LIN {X 0,Y 236.009,Z 217.756,A -85,B 0,C 180,E1 -19840.931,E2 -19840.931} C_VEL
LIN {X 0,Y 236.536,Z 220.925,A -85,B 0,C 180,E1 -19845.488,E2 -19845.488} C_VEL
LIN {X 0,Y 237.16,Z 224.354,A -85,B 0,C 180,E1 -19849.755,E2 -19849.755} C_VEL
LIN {X 0,Y 237.857,Z 228.006,A -85,B 0,C 180,E1 -19853.776,E2 -19853.776} C_VEL
LIN {X 0,Y 238.192,Z 230.1,A -85,B 0,C 180,E1 -19855.902,E2 -19855.902} C_VEL
LIN {X 0,Y 238.171,Z 231.141,A -85,B 0,C 180,E1 -19856.891,E2 -19856.891} C_VEL
LIN {X 0,Y 237.53,Z 232.457,A -85,B 0,C 180,E1 -19857.82,E2 -19857.82} C_VEL
LIN {X 0,Y 236.053,Z 234.265,A -85,B 0,C 180,E1 -19858.662,E2 -19858.662} C_VEL
LIN {X 0,Y 233.823,Z 237.363,A -85,B 0,C 180,E1 -19859.655,E2 -19859.655} C_VEL
LIN {X 0,Y 232.498,Z 240.8,A -85,B 0,C 180,E1 -19860.41,E2 -19860.41} C_VEL
LIN {X 0,Y 232.468,Z 243.65,A -85,B 0,C 180,E1 -19860.853,E2 -19860.853} C_VEL
LIN {X 0,Y 234.615,Z 253.264,A -85,B 0,C 180,E1 -19862.335,E2 -19862.335} C_VEL
LIN {X 0,Y 236.051,Z 263.876,A -85,B 0,C 180,E1 -19864.108,E2 -19864.108} C_VEL
LIN {X 0,Y 236.356,Z 273.236,A -85,B 0,C 180,E1 -19865.867,E2 -19865.867} C_VEL
LIN {X 0,Y 235.97,Z 280.551,A -85,B 0,C 180,E1 -19867.414,E2 -19867.414} C_VEL
LIN {X 0,Y 234.95,Z 287.098,A -85,B 0,C 180,E1 -19868.964,E2 -19868.964} C_VEL
LIN {X 0,Y 233.172,Z 293.307,A -85,B 0,C 180,E1 -19870.637,E2 -19870.637} C_VEL
LIN {X 0,Y 231.381,Z 298.539,A -85,B 0,C 180,E1 -19872.318,E2 -19872.318} C_VEL
LIN {X 0,Y 229.875,Z 302.919,A -85,B 0,C 180,E1 -19874.029,E2 -19874.029} C_VEL
LIN {X 0,Y 228.132,Z 308.12,A -85,B 0,C 180,E1 -19876.641,E2 -19876.641} C_VEL
LIN {X 0,Y 226.879,Z 311.977,A -85,B 0,C 180,E1 -19879.289,E2 -19879.289} C_VEL
LIN {X 0,Y 226.283,Z 313.766,A -85,B 0,C 180,E1 -19881.067,E2 -19881.067} C_VEL
LIN {X 0,Y 225.924,Z 315.065,A -85,B 0,C 180,E1 -19882.852,E2 -19882.852} C_VEL
LIN {X 0,Y 225.7,Z 316.017,A -85,B 0,C 180,E1 -19885.174,E2 -19885.174} C_VEL
LIN {X 0,Y 225.696,Z 316.253,A -85,B 0,C 180,E1 -19886.43,E2 -19886.43} C_VEL
LIN {X 0,Y 225.832,Z 316.034,A -85,B 0,C 180,E1 -19888.217,E2 -19888.217} C_VEL
LIN {X 0,Y 225.879,Z 315.278,A -85,B 0,C 180,E1 -19890,E2 -19890} C_VEL
LIN {X 0,Y 225.876,Z 314.017,A -85,B 0,C 180,E1 -19891.783,E2 -19891.783} C_VEL
LIN {X 0,Y 225.812,Z 311.128,A -85,B 0,C 180,E1 -19894.425,E2 -19894.425} C_VEL
LIN {X 0,Y 225.998,Z 306.803,A -85,B 0,C 180,E1 -19897.146,E2 -19897.146} C_VEL
LIN {X 0,Y 226.408,Z 301.952,A -85,B 0,C 180,E1 -19899.38,E2 -19899.38} C_VEL
LIN {X 0,Y 227.019,Z 295.755,A -85,B 0,C 180,E1 -19901.609,E2 -19901.609} C_VEL
LIN {X 0,Y 227.707,Z 289.678,A -85,B 0,C 180,E1 -19903.385,E2 -19903.385} C_VEL
LIN {X 0,Y 228.46,Z 283.285,A -85,B 0,C 180,E1 -19904.93,E2 -19904.93} C_VEL
LIN {X 0,Y 229.261,Z 278.016,A -85,B 0,C 180,E1 -19906.016,E2 -19906.016} C_VEL
LIN {X 0,Y 229.144,Z 270.13,A -85,B 0,C 180,E1 -19907.4,E2 -19907.4} C_VEL
LIN {X 0,Y 228.693,Z 261.091,A -85,B 0,C 180,E1 -19908.697,E2 -19908.697} C_VEL
LIN {X 0,Y 228.089,Z 252.419,A -85,B 0,C 180,E1 -19909.695,E2 -19909.695} C_VEL
LIN {X 0,Y 227.211,Z 241.832,A -85,B 0,C 180,E1 -19910.63,E2 -19910.63} C_VEL
LIN {X 0,Y 226.862,Z 237.785,A -85,B 0,C 180,E1 -19910.93,E2 -19910.93} C_VEL
LIN {X 0,Y 228.112,Z 230.392,A -85,B 0,C 180,E1 -19916.685,E2 -19916.685} C_VEL
LIN {X 0,Y 229.463,Z 224.432,A -85,B 0,C 180,E1 -19921.378,E2 -19921.378} C_VEL
LIN {X 0,Y 229.69,Z 223.191,A -85,B 0,C 180,E1 -19922.376,E2 -19922.376} C_VEL
LIN {X 0,Y 229.223,Z 219.34,A -85,B 0,C 180,E1 -19925.63,E2 -19925.63} C_VEL
LIN {X 0,Y 228.198,Z 214.067,A -85,B 0,C 180,E1 -19930.298,E2 -19930.298} C_VEL
LIN {X 0,Y 227.968,Z 212.904,A -85,B 0,C 180,E1 -19931.516,E2 -19931.516} C_VEL
LIN {X 0,Y 227.833,Z 212.914,A -85,B 0,C 180,E1 -19935.194,E2 -19935.194} C_VEL
LIN {X 0,Y 227.814,Z 212.918,A -85,B 0,C 180,E1 -19939.619,E2 -19939.619} C_VEL
LIN {X 0,Y 227.885,Z 212.91,A -85,B 0,C 180,E1 -19944.128,E2 -19944.128} C_VEL
LIN {X 0,Y 227.871,Z 212.913,A -85,B 0,C 180,E1 -19948.377,E2 -19948.377} C_VEL
LIN {X 0,Y 227.884,Z 212.907,A -85,B 0,C 180,E1 -19952.443,E2 -19952.443} C_VEL
LIN {X 0,Y 227.911,Z 212.907,A -85,B 0,C 180,E1 -19956.366,E2 -19956.366} C_VEL
LIN {X 0,Y 227.942,Z 212.901,A -85,B 0,C 180,E1 -19960.173,E2 -19960.173} C_VEL
LIN {X 0,Y 228.062,Z 212.889,A -85,B 0,C 180,E1 -19963.897,E2 -19963.897} C_VEL
LIN {X 0,Y 228.076,Z 212.888,A -85,B 0,C 180,E1 -19967.542,E2 -19967.542} C_VEL
LIN {X 0,Y 228.267,Z 212.861,A -85,B 0,C 180,E1 -19971.143,E2 -19971.143} C_VEL
LIN {X 0,Y 228.322,Z 212.855,A -85,B 0,C 180,E1 -19972.926,E2 -19972.926} C_VEL
LIN {X 0,Y 228.557,Z 212.822,A -85,B 0,C 180,E1 -19978.236,E2 -19978.236} C_VEL
LIN {X 0,Y 228.557,Z 212.826,A -85,B 0,C 180,E1 -19981.761,E2 -19981.761} C_VEL
LIN {X 0,Y 228.321,Z 212.856,A -85,B 0,C 180,E1 -19987.071,E2 -19987.071} C_VEL
LIN {X 0,Y 228.144,Z 212.879,A -85,B 0,C 180,E1 -19990.65,E2 -19990.65} C_VEL
LIN {X 0,Y 228.036,Z 212.89,A -85,B 0,C 180,E1 -19994.272,E2 -19994.272} C_VEL
LIN {X 0,Y 227.952,Z 212.901,A -85,B 0,C 180,E1 -19997.956,E2 -19997.956} C_VEL
LIN {X 0,Y 227.915,Z 212.907,A -85,B 0,C 180,E1 -20002.318,E2 -20002.318} C_VEL
LIN {X 0,Y 227.942,Z 212.905,A -85,B 0,C 180,E1 -20006.601,E2 -20006.601} C_VEL
LIN {X 0,Y 227.908,Z 212.908,A -85,B 0,C 180,E1 -20010.294,E2 -20010.294} C_VEL
LIN {X 0,Y 227.888,Z 212.908,A -85,B 0,C 180,E1 -20013.716,E2 -20013.716} C_VEL
LIN {X 0,Y 227.867,Z 212.914,A -85,B 0,C 180,E1 -20018.084,E2 -20018.084} C_VEL
LIN {X 0,Y 227.81,Z 212.919,A -85,B 0,C 180,E1 -20022.74,E2 -20022.74} C_VEL
LIN {X 0,Y 227.807,Z 212.918,A -85,B 0,C 180,E1 -20027.256,E2 -20027.256} C_VEL
LIN {X 0,Y 227.84,Z 212.918,A -85,B 0,C 180,E1 -20031.907,E2 -20031.907} C_VEL
LIN {X 0,Y 227.877,Z 212.907,A -85,B 0,C 180,E1 -20036.375,E2 -20036.375} C_VEL
LIN {X 0,Y 227.915,Z 212.906,A -85,B 0,C 180,E1 -20040.437,E2 -20040.437} C_VEL
LIN {X 0,Y 227.923,Z 212.902,A -85,B 0,C 180,E1 -20044.425,E2 -20044.425} C_VEL
LIN {X 0,Y 227.956,Z 212.9,A -85,B 0,C 180,E1 -20048.286,E2 -20048.286} C_VEL
LIN {X 0,Y 228.028,Z 212.891,A -85,B 0,C 180,E1 -20052.825,E2 -20052.825} C_VEL
LIN {X 0,Y 228.088,Z 212.885,A -85,B 0,C 180,E1 -20057.544,E2 -20057.544} C_VEL
LIN {X 0,Y 228.299,Z 212.857,A -85,B 0,C 180,E1 -20061.145,E2 -20061.145} C_VEL
LIN {X 0,Y 228.348,Z 212.852,A -85,B 0,C 180,E1 -20062.928,E2 -20062.928} C_VEL
LIN {X 0,Y 228.547,Z 212.827,A -85,B 0,C 180,E1 -20068.237,E2 -20068.237} C_VEL
LIN {X 0,Y 228.547,Z 212.825,A -85,B 0,C 180,E1 -20071.762,E2 -20071.762} C_VEL
LIN {X 0,Y 228.342,Z 212.851,A -85,B 0,C 180,E1 -20077.072,E2 -20077.072} C_VEL
LIN {X 0,Y 228.069,Z 212.889,A -85,B 0,C 180,E1 -20080.654,E2 -20080.654} C_VEL
LIN {X 0,Y 227.568,Z 212.948,A -85,B 0,C 180,E1 -20085.219,E2 -20085.219} C_VEL
LIN {X 0,Y 227.387,Z 213.262,A -85,B 0,C 180,E1 -20086.151,E2 -20086.151} C_VEL
LIN {X 0,Y 226.732,Z 218.382,A -85,B 0,C 180,E1 -20091.836,E2 -20091.836} C_VEL
LIN {X 0,Y 226.515,Z 221.365,A -85,B 0,C 180,E1 -20095.069,E2 -20095.069} C_VEL
LIN {X 0,Y 228.367,Z 233.039,A -85,B 0,C 180,E1 -20096.142,E2 -20096.142} C_VEL
LIN {X 0,Y 229.539,Z 241.029,A -85,B 0,C 180,E1 -20097.094,E2 -20097.094} C_VEL
LIN {X 0,Y 230.39,Z 248.198,A -85,B 0,C 180,E1 -20098.118,E2 -20098.118} C_VEL
LIN {X 0,Y 230.632,Z 251.482,A -85,B 0,C 180,E1 -20098.632,E2 -20098.632} C_VEL
LIN {X 0,Y 229.569,Z 260.933,A -85,B 0,C 180,E1 -20100.34,E2 -20100.34} C_VEL
LIN {X 0,Y 228.561,Z 268.372,A -85,B 0,C 180,E1 -20102.033,E2 -20102.033} C_VEL
LIN {X 0,Y 227.799,Z 274.475,A -85,B 0,C 180,E1 -20103.733,E2 -20103.733} C_VEL
LIN {X 0,Y 226.95,Z 281.168,A -85,B 0,C 180,E1 -20106.042,E2 -20106.042} C_VEL
LIN {X 0,Y 226.266,Z 286.441,A -85,B 0,C 180,E1 -20108.405,E2 -20108.405} C_VEL
LIN {X 0,Y 225.798,Z 290.425,A -85,B 0,C 180,E1 -20110.815,E2 -20110.815} C_VEL
LIN {X 0,Y 225.52,Z 294.234,A -85,B 0,C 180,E1 -20114.215,E2 -20114.215} C_VEL
LIN {X 0,Y 225.654,Z 295.712,A -85,B 0,C 180,E1 -20116.752,E2 -20116.752} C_VEL
LIN {X 0,Y 226.034,Z 296.092,A -85,B 0,C 180,E1 -20119.238,E2 -20119.238} C_VEL
LIN {X 0,Y 226.727,Z 295.476,A -85,B 0,C 180,E1 -20121.69,E2 -20121.69} C_VEL
LIN {X 0,Y 227.729,Z 293.88,A -85,B 0,C 180,E1 -20124.103,E2 -20124.103} C_VEL
LIN {X 0,Y 228.965,Z 291.312,A -85,B 0,C 180,E1 -20126.463,E2 -20126.463} C_VEL
LIN {X 0,Y 230.971,Z 286.624,A -85,B 0,C 180,E1 -20129.36,E2 -20129.36} C_VEL
LIN {X 0,Y 233.004,Z 281.169,A -85,B 0,C 180,E1 -20131.726,E2 -20131.726} C_VEL
LIN {X 0,Y 234.562,Z 276.653,A -85,B 0,C 180,E1 -20133.295,E2 -20133.295} C_VEL
LIN {X 0,Y 236.617,Z 270.345,A -85,B 0,C 180,E1 -20135.063,E2 -20135.063} C_VEL
LIN {X 0,Y 238.257,Z 264.393,A -85,B 0,C 180,E1 -20136.444,E2 -20136.444} C_VEL
LIN {X 0,Y 237.992,Z 256.862,A -85,B 0,C 180,E1 -20138.222,E2 -20138.222} C_VEL
LIN {X 0,Y 236.795,Z 248.433,A -85,B 0,C 180,E1 -20140.045,E2 -20140.045} C_VEL
LIN {X 0,Y 234.593,Z 239.575,A -85,B 0,C 180,E1 -20141.832,E2 -20141.832} C_VEL
LIN {X 0,Y 230.936,Z 229.569,A -85,B 0,C 180,E1 -20143.742,E2 -20143.742} C_VEL
LIN {X 0,Y 229.933,Z 227.141,A -85,B 0,C 180,E1 -20144.205,E2 -20144.205} C_VEL
LIN {X 0,Y 228.809,Z 223.879,A -85,B 0,C 180,E1 -20144.81,E2 -20144.81} C_VEL
LIN {X 0,Y 229.302,Z 220.946,A -85,B 0,C 180,E1 -20149.405,E2 -20149.405} C_VEL
LIN {X 0,Y 229.234,Z 218.974,A -85,B 0,C 180,E1 -20152.957,E2 -20152.957} C_VEL
LIN {X 0,Y 229.128,Z 216.447,A -85,B 0,C 180,E1 -20158.244,E2 -20158.244} C_VEL
LIN {X 0,Y 229.155,Z 215.721,A -85,B 0,C 180,E1 -20160.002,E2 -20160.002} C_VEL
LIN {X 0,Y 228.593,Z 214.576,A -85,B 0,C 180,E1 -20163.527,E2 -20163.527} C_VEL
LIN {X 0,Y 228.444,Z 213.575,A -85,B 0,C 180,E1 -20167.07,E2 -20167.07} C_VEL
LIN {X 0,Y 228.147,Z 212.893,A -85,B 0,C 180,E1 -20170.653,E2 -20170.653} C_VEL
LIN {X 0,Y 228.066,Z 212.889,A -85,B 0,C 180,E1 -20174.273,E2 -20174.273} C_VEL
LIN {X 0,Y 228.006,Z 212.896,A -85,B 0,C 180,E1 -20177.954,E2 -20177.954} C_VEL
LIN {X 0,Y 227.933,Z 212.905,A -85,B 0,C 180,E1 -20182.331,E2 -20182.331} C_VEL
LIN {X 0,Y 228.046,Z 213.463,A -85,B 0,C 180,E1 -20186.655,E2 -20186.655} C_VEL
LIN {X 0,Y 228.219,Z 214.544,A -85,B 0,C 180,E1 -20190.429,E2 -20190.429} C_VEL
LIN {X 0,Y 228.472,Z 215.839,A -85,B 0,C 180,E1 -20193.846,E2 -20193.846} C_VEL
LIN {X 0,Y 228.798,Z 217.794,A -85,B 0,C 180,E1 -20197.905,E2 -20197.905} C_VEL
LIN {X 0,Y 229.049,Z 219.022,A -85,B 0,C 180,E1 -20200.119,E2 -20200.119} C_VEL
LIN {X 0,Y 229.547,Z 222.05,A -85,B 0,C 180,E1 -20204.765,E2 -20204.765} C_VEL
LIN {X 0,Y 229.969,Z 224.284,A -85,B 0,C 180,E1 -20207.753,E2 -20207.753} C_VEL
LIN {X 0,Y 230.669,Z 228.186,A -85,B 0,C 180,E1 -20212.39,E2 -20212.39} C_VEL
LIN {X 0,Y 231.105,Z 230.795,A -85,B 0,C 180,E1 -20215.195,E2 -20215.195} C_VEL
LIN {X 0,Y 231.186,Z 232.43,A -85,B 0,C 180,E1 -20216.826,E2 -20216.826} C_VEL
LIN {X 0,Y 230.299,Z 235.782,A -85,B 0,C 180,E1 -20219.736,E2 -20219.736} C_VEL
LIN {X 0,Y 231.26,Z 239.321,A -85,B 0,C 180,E1 -20220.208,E2 -20220.208} C_VEL
LIN {X 0,Y 232.468,Z 243.65,A -85,B 0,C 180,E1 -20220.853,E2 -20220.853} C_VEL
LIN {X 0,Y 232.865,Z 248.996,A -85,B 0,C 180,E1 -20221.485,E2 -20221.485} C_VEL
LIN {X 0,Y 231.841,Z 258.038,A -85,B 0,C 180,E1 -20222.481,E2 -20222.481} C_VEL
LIN {X 0,Y 230.335,Z 266.707,A -85,B 0,C 180,E1 -20223.644,E2 -20223.644} C_VEL
LIN {X 0,Y 229.968,Z 271.47,A -85,B 0,C 180,E1 -20224.529,E2 -20224.529} C_VEL
LIN {X 0,Y 229.709,Z 278.727,A -85,B 0,C 180,E1 -20226.085,E2 -20226.085} C_VEL
LIN {X 0,Y 228.639,Z 286.775,A -85,B 0,C 180,E1 -20228.06,E2 -20228.06} C_VEL
LIN {X 0,Y 227.007,Z 292.445,A -85,B 0,C 180,E1 -20229.617,E2 -20229.617} C_VEL
LIN {X 0,Y 225.068,Z 297.746,A -85,B 0,C 180,E1 -20231.333,E2 -20231.333} C_VEL
LIN {X 0,Y 223.058,Z 303.147,A -85,B 0,C 180,E1 -20233.527,E2 -20233.527} C_VEL
LIN {X 0,Y 221.776,Z 306.677,A -85,B 0,C 180,E1 -20235.315,E2 -20235.315} C_VEL
LIN {X 0,Y 220.267,Z 310.783,A -85,B 0,C 180,E1 -20238.031,E2 -20238.031} C_VEL
LIN {X 0,Y 219.251,Z 313.662,A -85,B 0,C 180,E1 -20240.778,E2 -20240.778} C_VEL
LIN {X 0,Y 218.861,Z 314.868,A -85,B 0,C 180,E1 -20242.62,E2 -20242.62} C_VEL
LIN {X 0,Y 218.602,Z 315.795,A -85,B 0,C 180,E1 -20245.315,E2 -20245.315} C_VEL
LIN {X 0,Y 218.759,Z 315.646,A -85,B 0,C 180,E1 -20248.159,E2 -20248.159} C_VEL
LIN {X 0,Y 218.811,Z 314.813,A -85,B 0,C 180,E1 -20250,E2 -20250} C_VEL
LIN {X 0,Y 218.809,Z 313.465,A -85,B 0,C 180,E1 -20251.841,E2 -20251.841} C_VEL
LIN {X 0,Y 218.775,Z 311.577,A -85,B 0,C 180,E1 -20253.684,E2 -20253.684} C_VEL
LIN {X 0,Y 218.774,Z 309.105,A -85,B 0,C 180,E1 -20255.531,E2 -20255.531} C_VEL
LIN {X 0,Y 218.943,Z 305.998,A -85,B 0,C 180,E1 -20257.377,E2 -20257.377} C_VEL
LIN {X 0,Y 219.395,Z 301.004,A -85,B 0,C 180,E1 -20259.682,E2 -20259.682} C_VEL
LIN {X 0,Y 219.854,Z 296.084,A -85,B 0,C 180,E1 -20261.525,E2 -20261.525} C_VEL
LIN {X 0,Y 220.575,Z 290.142,A -85,B 0,C 180,E1 -20263.356,E2 -20263.356} C_VEL
LIN {X 0,Y 221.6,Z 281.884,A -85,B 0,C 180,E1 -20265.404,E2 -20265.404} C_VEL
LIN {X 0,Y 222.223,Z 277.593,A -85,B 0,C 180,E1 -20266.301,E2 -20266.301} C_VEL
LIN {X 0,Y 222.037,Z 269.274,A -85,B 0,C 180,E1 -20267.798,E2 -20267.798} C_VEL
LIN {X 0,Y 221.668,Z 261.438,A -85,B 0,C 180,E1 -20268.965,E2 -20268.965} C_VEL
LIN {X 0,Y 221.104,Z 253.058,A -85,B 0,C 180,E1 -20269.981,E2 -20269.981} C_VEL
LIN {X 0,Y 220.373,Z 243.847,A -85,B 0,C 180,E1 -20270.852,E2 -20270.852} C_VEL
LIN {X 0,Y 219.832,Z 237.551,A -85,B 0,C 180,E1 -20271.327,E2 -20271.327} C_VEL
LIN {X 0,Y 221.123,Z 230.359,A -85,B 0,C 180,E1 -20277.133,E2 -20277.133} C_VEL
LIN {X 0,Y 222.375,Z 225.098,A -85,B 0,C 180,E1 -20281.424,E2 -20281.424} C_VEL
LIN {X 0,Y 222.634,Z 223.84,A -85,B 0,C 180,E1 -20282.456,E2 -20282.456} C_VEL
LIN {X 0,Y 222.134,Z 219.983,A -85,B 0,C 180,E1 -20285.825,E2 -20285.825} C_VEL
LIN {X 0,Y 221.036,Z 214.344,A -85,B 0,C 180,E1 -20291.028,E2 -20291.028} C_VEL
LIN {X 0,Y 220.908,Z 213.784,A -85,B 0,C 180,E1 -20291.704,E2 -20291.704} C_VEL
LIN {X 0,Y 220.773,Z 213.793,A -85,B 0,C 180,E1 -20295.544,E2 -20295.544} C_VEL
LIN {X 0,Y 220.789,Z 213.796,A -85,B 0,C 180,E1 -20300.458,E2 -20300.458} C_VEL
LIN {X 0,Y 220.829,Z 213.788,A -85,B 0,C 180,E1 -20302.792,E2 -20302.792} C_VEL
LIN {X 0,Y 220.821,Z 213.789,A -85,B 0,C 180,E1 -20307.243,E2 -20307.243} C_VEL
LIN {X 0,Y 220.832,Z 213.788,A -85,B 0,C 180,E1 -20311.484,E2 -20311.484} C_VEL
LIN {X 0,Y 220.867,Z 213.784,A -85,B 0,C 180,E1 -20315.564,E2 -20315.564} C_VEL
LIN {X 0,Y 220.889,Z 213.783,A -85,B 0,C 180,E1 -20319.512,E2 -20319.512} C_VEL
LIN {X 0,Y 221.021,Z 213.764,A -85,B 0,C 180,E1 -20323.369,E2 -20323.369} C_VEL
LIN {X 0,Y 221.016,Z 213.766,A -85,B 0,C 180,E1 -20327.137,E2 -20327.137} C_VEL
LIN {X 0,Y 221.205,Z 213.739,A -85,B 0,C 180,E1 -20330.858,E2 -20330.858} C_VEL
LIN {X 0,Y 221.139,Z 213.75,A -85,B 0,C 180,E1 -20334.527,E2 -20334.527} C_VEL
LIN {X 0,Y 221.515,Z 213.699,A -85,B 0,C 180,E1 -20338.18,E2 -20338.18} C_VEL
LIN {X 0,Y 221.514,Z 213.703,A -85,B 0,C 180,E1 -20341.817,E2 -20341.817} C_VEL
LIN {X 0,Y 221.257,Z 213.735,A -85,B 0,C 180,E1 -20347.298,E2 -20347.298} C_VEL
LIN {X 0,Y 221.064,Z 213.762,A -85,B 0,C 180,E1 -20350.995,E2 -20350.995} C_VEL
LIN {X 0,Y 220.978,Z 213.77,A -85,B 0,C 180,E1 -20356.631,E2 -20356.631} C_VEL
LIN {X 0,Y 220.874,Z 213.786,A -85,B 0,C 180,E1 -20360.486,E2 -20360.486} C_VEL
LIN {X 0,Y 220.862,Z 213.784,A -85,B 0,C 180,E1 -20364.434,E2 -20364.434} C_VEL
LIN {X 0,Y 220.836,Z 213.79,A -85,B 0,C 180,E1 -20368.512,E2 -20368.512} C_VEL
LIN {X 0,Y 220.823,Z 213.789,A -85,B 0,C 180,E1 -20372.753,E2 -20372.753} C_VEL
LIN {X 0,Y 220.836,Z 213.787,A -85,B 0,C 180,E1 -20377.286,E2 -20377.286} C_VEL
LIN {X 0,Y 220.772,Z 213.797,A -85,B 0,C 180,E1 -20381.949,E2 -20381.949} C_VEL
LIN {X 0,Y 220.77,Z 213.797,A -85,B 0,C 180,E1 -20385.544,E2 -20385.544} C_VEL
LIN {X 0,Y 220.802,Z 213.791,A -85,B 0,C 180,E1 -20390.462,E2 -20390.462} C_VEL
LIN {X 0,Y 220.799,Z 213.792,A -85,B 0,C 180,E1 -20395.044,E2 -20395.044} C_VEL
LIN {X 0,Y 220.863,Z 213.786,A -85,B 0,C 180,E1 -20399.394,E2 -20399.394} C_VEL
LIN {X 0,Y 220.89,Z 213.781,A -85,B 0,C 180,E1 -20403.548,E2 -20403.548} C_VEL
LIN {X 0,Y 220.872,Z 213.785,A -85,B 0,C 180,E1 -20407.552,E2 -20407.552} C_VEL
LIN {X 0,Y 220.978,Z 213.768,A -85,B 0,C 180,E1 -20412.57,E2 -20412.57} C_VEL
LIN {X 0,Y 221.02,Z 213.768,A -85,B 0,C 180,E1 -20417.139,E2 -20417.139} C_VEL
LIN {X 0,Y 221.23,Z 213.74,A -85,B 0,C 180,E1 -20420.86,E2 -20420.86} C_VEL
LIN {X 0,Y 221.283,Z 213.731,A -85,B 0,C 180,E1 -20422.701,E2 -20422.701} C_VEL
LIN {X 0,Y 221.505,Z 213.704,A -85,B 0,C 180,E1 -20428.181,E2 -20428.181} C_VEL
LIN {X 0,Y 221.506,Z 213.703,A -85,B 0,C 180,E1 -20431.818,E2 -20431.818} C_VEL
LIN {X 0,Y 221.272,Z 213.731,A -85,B 0,C 180,E1 -20437.299,E2 -20437.299} C_VEL
LIN {X 0,Y 220.987,Z 213.769,A -85,B 0,C 180,E1 -20441,E2 -20441} C_VEL
LIN {X 0,Y 220.411,Z 213.84,A -85,B 0,C 180,E1 -20445.725,E2 -20445.725} C_VEL
LIN {X 0,Y 219.758,Z 218.002,A -85,B 0,C 180,E1 -20450.596,E2 -20450.596} C_VEL
LIN {X 0,Y 219.478,Z 221.64,A -85,B 0,C 180,E1 -20454.663,E2 -20454.663} C_VEL
LIN {X 0,Y 221.167,Z 232.252,A -85,B 0,C 180,E1 -20455.655,E2 -20455.655} C_VEL
LIN {X 0,Y 222.461,Z 241.134,A -85,B 0,C 180,E1 -20456.73,E2 -20456.73} C_VEL
LIN {X 0,Y 223.422,Z 249.392,A -85,B 0,C 180,E1 -20457.957,E2 -20457.957} C_VEL
LIN {X 0,Y 223.475,Z 253.385,A -85,B 0,C 180,E1 -20458.607,E2 -20458.607} C_VEL
LIN {X 0,Y 222.354,Z 262.471,A -85,B 0,C 180,E1 -20460.379,E2 -20460.379} C_VEL
LIN {X 0,Y 221.491,Z 268.807,A -85,B 0,C 180,E1 -20461.892,E2 -20461.892} C_VEL
LIN {X 0,Y 220.671,Z 275.229,A -85,B 0,C 180,E1 -20463.756,E2 -20463.756} C_VEL
LIN {X 0,Y 219.861,Z 281.369,A -85,B 0,C 180,E1 -20465.956,E2 -20465.956} C_VEL
LIN {X 0,Y 219.123,Z 286.942,A -85,B 0,C 180,E1 -20468.543,E2 -20468.543} C_VEL
LIN {X 0,Y 218.655,Z 290.998,A -85,B 0,C 180,E1 -20471.118,E2 -20471.118} C_VEL
LIN {X 0,Y 218.478,Z 292.751,A -85,B 0,C 180,E1 -20472.495,E2 -20472.495} C_VEL
LIN {X 0,Y 218.455,Z 294.983,A -85,B 0,C 180,E1 -20475.054,E2 -20475.054} C_VEL
LIN {X 0,Y 218.658,Z 296.19,A -85,B 0,C 180,E1 -20477.668,E2 -20477.668} C_VEL
LIN {X 0,Y 219.199,Z 296.352,A -85,B 0,C 180,E1 -20480.308,E2 -20480.308} C_VEL
LIN {X 0,Y 220.122,Z 295.442,A -85,B 0,C 180,E1 -20482.958,E2 -20482.958} C_VEL
LIN {X 0,Y 221.399,Z 293.41,A -85,B 0,C 180,E1 -20485.622,E2 -20485.622} C_VEL
LIN {X 0,Y 223.037,Z 290.008,A -85,B 0,C 180,E1 -20488.297,E2 -20488.297} C_VEL
LIN {X 0,Y 224.705,Z 286.115,A -85,B 0,C 180,E1 -20490.501,E2 -20490.501} C_VEL
LIN {X 0,Y 226.298,Z 282.229,A -85,B 0,C 180,E1 -20492.237,E2 -20492.237} C_VEL
LIN {X 0,Y 228.131,Z 277.276,A -85,B 0,C 180,E1 -20494.03,E2 -20494.03} C_VEL
LIN {X 0,Y 230.295,Z 271.021,A -85,B 0,C 180,E1 -20495.839,E2 -20495.839} C_VEL
LIN {X 0,Y 231.776,Z 266.166,A -85,B 0,C 180,E1 -20497.022,E2 -20497.022} C_VEL
LIN {X 0,Y 231.728,Z 259.741,A -85,B 0,C 180,E1 -20498.659,E2 -20498.659} C_VEL
LIN {X 0,Y 230.892,Z 252.127,A -85,B 0,C 180,E1 -20500.44,E2 -20500.44} C_VEL
LIN {X 0,Y 229.222,Z 244.359,A -85,B 0,C 180,E1 -20502.147,E2 -20502.147} C_VEL
LIN {X 0,Y 226.84,Z 236.486,A -85,B 0,C 180,E1 -20503.811,E2 -20503.811} C_VEL
LIN {X 0,Y 223.811,Z 228.52,A -85,B 0,C 180,E1 -20505.452,E2 -20505.452} C_VEL
LIN {X 0,Y 222.232,Z 225.386,A -85,B 0,C 180,E1 -20506.165,E2 -20506.165} C_VEL
LIN {X 0,Y 221.993,Z 224.25,A -85,B 0,C 180,E1 -20506.383,E2 -20506.383} C_VEL
LIN {X 0,Y 222.329,Z 222.625,A -85,B 0,C 180,E1 -20509.068,E2 -20509.068} C_VEL
LIN {X 0,Y 222.296,Z 220.642,A -85,B 0,C 180,E1 -20512.736,E2 -20512.736} C_VEL
LIN {X 0,Y 222.237,Z 218.137,A -85,B 0,C 180,E1 -20518.189,E2 -20518.189} C_VEL
LIN {X 0,Y 222.252,Z 217.404,A -85,B 0,C 180,E1 -20520.002,E2 -20520.002} C_VEL
LIN {X 0,Y 222.066,Z 216.782,A -85,B 0,C 180,E1 -20521.815,E2 -20521.815} C_VEL
LIN {X 0,Y 221.554,Z 215.343,A -85,B 0,C 180,E1 -20527.291,E2 -20527.291} C_VEL
LIN {X 0,Y 221.272,Z 214.705,A -85,B 0,C 180,E1 -20530.988,E2 -20530.988} C_VEL
LIN {X 0,Y 221.104,Z 214.351,A -85,B 0,C 180,E1 -20534.733,E2 -20534.733} C_VEL
LIN {X 0,Y 221.01,Z 214.32,A -85,B 0,C 180,E1 -20538.543,E2 -20538.543} C_VEL
LIN {X 0,Y 221.041,Z 214.683,A -85,B 0,C 180,E1 -20542.772,E2 -20542.772} C_VEL
LIN {X 0,Y 221.227,Z 215.514,A -85,B 0,C 180,E1 -20547.188,E2 -20547.188} C_VEL
LIN {X 0,Y 221.416,Z 216.643,A -85,B 0,C 180,E1 -20551.018,E2 -20551.018} C_VEL
LIN {X 0,Y 221.689,Z 218.119,A -85,B 0,C 180,E1 -20554.796,E2 -20554.796} C_VEL
LIN {X 0,Y 221.926,Z 219.47,A -85,B 0,C 180,E1 -20557.655,E2 -20557.655} C_VEL
LIN {X 0,Y 222.281,Z 221.687,A -85,B 0,C 180,E1 -20561.605,E2 -20561.605} C_VEL
LIN {X 0,Y 222.789,Z 224.649,A -85,B 0,C 180,E1 -20566.053,E2 -20566.053} C_VEL
LIN {X 0,Y 223.214,Z 226.933,A -85,B 0,C 180,E1 -20569.084,E2 -20569.084} C_VEL
LIN {X 0,Y 223.901,Z 230.535,A -85,B 0,C 180,E1 -20573.389,E2 -20573.389} C_VEL
LIN {X 0,Y 224.193,Z 233.673,A -85,B 0,C 180,E1 -20576.73,E2 -20576.73} C_VEL
LIN {X 0,Y 223.798,Z 235.454,A -85,B 0,C 180,E1 -20578.285,E2 -20578.285} C_VEL
LIN {X 0,Y 224.736,Z 238.836,A -85,B 0,C 180,E1 -20578.783,E2 -20578.783} C_VEL
LIN {X 0,Y 227.717,Z 250.379,A -85,B 0,C 180,E1 -20580.677,E2 -20580.677} C_VEL
LIN {X 0,Y 229.263,Z 259.707,A -85,B 0,C 180,E1 -20582.291,E2 -20582.291} C_VEL
LIN {X 0,Y 229.949,Z 269.59,A -85,B 0,C 180,E1 -20584.142,E2 -20584.142} C_VEL
LIN {X 0,Y 229.968,Z 271.47,A -85,B 0,C 180,E1 -20584.529,E2 -20584.529} C_VEL
LIN {X 0,Y 229.292,Z 276.264,A -85,B 0,C 180,E1 -20585.45,E2 -20585.45} C_VEL
LIN {X 0,Y 227.53,Z 280.938,A -85,B 0,C 180,E1 -20586.297,E2 -20586.297} C_VEL
LIN {X 0,Y 222.626,Z 289.438,A -85,B 0,C 180,E1 -20588.043,E2 -20588.043} C_VEL
LIN {X 0,Y 219.824,Z 294.488,A -85,B 0,C 180,E1 -20589.443,E2 -20589.443} C_VEL
LIN {X 0,Y 217.11,Z 301.491,A -85,B 0,C 180,E1 -20592.09,E2 -20592.09} C_VEL
LIN {X 0,Y 215.575,Z 305.274,A -85,B 0,C 180,E1 -20593.913,E2 -20593.913} C_VEL
LIN {X 0,Y 213.798,Z 309.622,A -85,B 0,C 180,E1 -20596.697,E2 -20596.697} C_VEL
LIN {X 0,Y 212.908,Z 311.875,A -85,B 0,C 180,E1 -20598.577,E2 -20598.577} C_VEL
LIN {X 0,Y 212.239,Z 313.56,A -85,B 0,C 180,E1 -20600.47,E2 -20600.47} C_VEL
LIN {X 0,Y 211.822,Z 314.672,A -85,B 0,C 180,E1 -20602.374,E2 -20602.374} C_VEL
LIN {X 0,Y 211.517,Z 315.549,A -85,B 0,C 180,E1 -20605.428,E2 -20605.428} C_VEL
LIN {X 0,Y 211.687,Z 315.215,A -85,B 0,C 180,E1 -20608.098,E2 -20608.098} C_VEL
LIN {X 0,Y 211.743,Z 314.342,A -85,B 0,C 180,E1 -20610,E2 -20610} C_VEL
LIN {X 0,Y 211.742,Z 312.897,A -85,B 0,C 180,E1 -20611.902,E2 -20611.902} C_VEL
LIN {X 0,Y 211.699,Z 309.213,A -85,B 0,C 180,E1 -20615.152,E2 -20615.152} C_VEL
LIN {X 0,Y 211.912,Z 305.101,A -85,B 0,C 180,E1 -20617.624,E2 -20617.624} C_VEL
LIN {X 0,Y 212.367,Z 299.976,A -85,B 0,C 180,E1 -20620.006,E2 -20620.006} C_VEL
LIN {X 0,Y 212.899,Z 294.924,A -85,B 0,C 180,E1 -20621.907,E2 -20621.907} C_VEL
LIN {X 0,Y 213.633,Z 288.818,A -85,B 0,C 180,E1 -20623.799,E2 -20623.799} C_VEL
LIN {X 0,Y 214.428,Z 282.389,A -85,B 0,C 180,E1 -20625.445,E2 -20625.445} C_VEL
LIN {X 0,Y 215.172,Z 277.051,A -85,B 0,C 180,E1 -20626.607,E2 -20626.607} C_VEL
LIN {X 0,Y 214.919,Z 268.607,A -85,B 0,C 180,E1 -20628.167,E2 -20628.167} C_VEL
LIN {X 0,Y 214.567,Z 260.69,A -85,B 0,C 180,E1 -20629.369,E2 -20629.369} C_VEL
LIN {X 0,Y 214.018,Z 252.164,A -85,B 0,C 180,E1 -20630.421,E2 -20630.421} C_VEL
LIN {X 0,Y 213.192,Z 241.514,A -85,B 0,C 180,E1 -20631.431,E2 -20631.431} C_VEL
LIN {X 0,Y 212.818,Z 237.297,A -85,B 0,C 180,E1 -20631.767,E2 -20631.767} C_VEL
LIN {X 0,Y 214.138,Z 230.317,A -85,B 0,C 180,E1 -20637.606,E2 -20637.606} C_VEL
LIN {X 0,Y 215.425,Z 225.134,A -85,B 0,C 180,E1 -20641.979,E2 -20641.979} C_VEL
LIN {X 0,Y 215.469,Z 223.207,A -85,B 0,C 180,E1 -20643.676,E2 -20643.676} C_VEL
LIN {X 0,Y 214.802,Z 219.488,A -85,B 0,C 180,E1 -20647.093,E2 -20647.093} C_VEL
LIN {X 0,Y 213.856,Z 214.661,A -85,B 0,C 180,E1 -20651.878,E2 -20651.878} C_VEL
LIN {X 0,Y 213.707,Z 214.675,A -85,B 0,C 180,E1 -20656.344,E2 -20656.344} C_VEL
LIN {X 0,Y 213.713,Z 214.674,A -85,B 0,C 180,E1 -20659.145,E2 -20659.145} C_VEL
LIN {X 0,Y 213.748,Z 214.67,A -85,B 0,C 180,E1 -20663.711,E2 -20663.711} C_VEL
LIN {X 0,Y 213.772,Z 214.67,A -85,B 0,C 180,E1 -20668.262,E2 -20668.262} C_VEL
LIN {X 0,Y 213.831,Z 214.657,A -85,B 0,C 180,E1 -20672.602,E2 -20672.602} C_VEL
LIN {X 0,Y 213.824,Z 214.661,A -85,B 0,C 180,E1 -20676.973,E2 -20676.973} C_VEL
LIN {X 0,Y 213.948,Z 214.643,A -85,B 0,C 180,E1 -20682.802,E2 -20682.802} C_VEL
LIN {X 0,Y 213.957,Z 214.644,A -85,B 0,C 180,E1 -20686.705,E2 -20686.705} C_VEL
LIN {X 0,Y 214.143,Z 214.618,A -85,B 0,C 180,E1 -20690.554,E2 -20690.554} C_VEL
LIN {X 0,Y 214.101,Z 214.626,A -85,B 0,C 180,E1 -20694.347,E2 -20694.347} C_VEL
LIN {X 0,Y 214.448,Z 214.579,A -85,B 0,C 180,E1 -20698.12,E2 -20698.12} C_VEL
LIN {X 0,Y 214.549,Z 214.57,A -85,B 0,C 180,E1 -20699.998,E2 -20699.998} C_VEL
LIN {X 0,Y 214.448,Z 214.583,A -85,B 0,C 180,E1 -20701.876,E2 -20701.876} C_VEL
LIN {X 0,Y 214.196,Z 214.613,A -85,B 0,C 180,E1 -20707.54,E2 -20707.54} C_VEL
LIN {X 0,Y 213.994,Z 214.64,A -85,B 0,C 180,E1 -20711.363,E2 -20711.363} C_VEL
LIN {X 0,Y 213.901,Z 214.65,A -85,B 0,C 180,E1 -20715.237,E2 -20715.237} C_VEL
LIN {X 0,Y 213.813,Z 214.663,A -85,B 0,C 180,E1 -20719.188,E2 -20719.188} C_VEL
LIN {X 0,Y 213.81,Z 214.659,A -85,B 0,C 180,E1 -20723.229,E2 -20723.229} C_VEL
LIN {X 0,Y 213.828,Z 214.66,A -85,B 0,C 180,E1 -20727.448,E2 -20727.448} C_VEL
LIN {X 0,Y 213.778,Z 214.664,A -85,B 0,C 180,E1 -20731.734,E2 -20731.734} C_VEL
LIN {X 0,Y 213.75,Z 214.673,A -85,B 0,C 180,E1 -20736.285,E2 -20736.285} C_VEL
LIN {X 0,Y 213.713,Z 214.672,A -85,B 0,C 180,E1 -20741.122,E2 -20741.122} C_VEL
LIN {X 0,Y 213.704,Z 214.677,A -85,B 0,C 180,E1 -20743.676,E2 -20743.676} C_VEL
LIN {X 0,Y 213.702,Z 214.676,A -85,B 0,C 180,E1 -20746.342,E2 -20746.342} C_VEL
LIN {X 0,Y 213.713,Z 214.672,A -85,B 0,C 180,E1 -20749.141,E2 -20749.141} C_VEL
LIN {X 0,Y 213.74,Z 214.674,A -85,B 0,C 180,E1 -20753.71,E2 -20753.71} C_VEL
LIN {X 0,Y 213.79,Z 214.664,A -85,B 0,C 180,E1 -20758.723,E2 -20758.723} C_VEL
LIN {X 0,Y 213.821,Z 214.661,A -85,B 0,C 180,E1 -20762.602,E2 -20762.602} C_VEL
LIN {X 0,Y 213.846,Z 214.658,A -85,B 0,C 180,E1 -20766.952,E2 -20766.952} C_VEL
LIN {X 0,Y 213.937,Z 214.646,A -85,B 0,C 180,E1 -20772.803,E2 -20772.803} C_VEL
LIN {X 0,Y 213.974,Z 214.643,A -85,B 0,C 180,E1 -20776.708,E2 -20776.708} C_VEL
LIN {X 0,Y 214.161,Z 214.619,A -85,B 0,C 180,E1 -20780.556,E2 -20780.556} C_VEL
LIN {X 0,Y 214.221,Z 214.609,A -85,B 0,C 180,E1 -20782.459,E2 -20782.459} C_VEL
LIN {X 0,Y 214.438,Z 214.584,A -85,B 0,C 180,E1 -20788.121,E2 -20788.121} C_VEL
LIN {X 0,Y 214.543,Z 214.569,A -85,B 0,C 180,E1 -20790,E2 -20790} C_VEL
LIN {X 0,Y 214.439,Z 214.583,A -85,B 0,C 180,E1 -20791.878,E2 -20791.878} C_VEL
LIN {X 0,Y 214.207,Z 214.611,A -85,B 0,C 180,E1 -20797.541,E2 -20797.541} C_VEL
LIN {X 0,Y 213.884,Z 214.653,A -85,B 0,C 180,E1 -20801.37,E2 -20801.37} C_VEL
LIN {X 0,Y 213.307,Z 214.775,A -85,B 0,C 180,E1 -20805.967,E2 -20805.967} C_VEL
LIN {X 0,Y 212.646,Z 219.391,A -85,B 0,C 180,E1 -20811.318,E2 -20811.318} C_VEL
LIN {X 0,Y 212.387,Z 221.931,A -85,B 0,C 180,E1 -20814.238,E2 -20814.238} C_VEL
LIN {X 0,Y 214.127,Z 232.487,A -85,B 0,C 180,E1 -20815.257,E2 -20815.257} C_VEL
LIN {X 0,Y 215.42,Z 241.533,A -85,B 0,C 180,E1 -20816.392,E2 -20816.392} C_VEL
LIN {X 0,Y 216.328,Z 248.963,A -85,B 0,C 180,E1 -20817.527,E2 -20817.527} C_VEL
LIN {X 0,Y 216.495,Z 253.581,A -85,B 0,C 180,E1 -20818.304,E2 -20818.304} C_VEL
LIN {X 0,Y 215.333,Z 262.638,A -85,B 0,C 180,E1 -20820.119,E2 -20820.119} C_VEL
LIN {X 0,Y 214.333,Z 269.872,A -85,B 0,C 180,E1 -20821.92,E2 -20821.92} C_VEL
LIN {X 0,Y 213.428,Z 276.772,A -85,B 0,C 180,E1 -20824.041,E2 -20824.041} C_VEL
LIN {X 0,Y 212.548,Z 283.127,A -85,B 0,C 180,E1 -20826.525,E2 -20826.525} C_VEL
LIN {X 0,Y 211.897,Z 288.054,A -85,B 0,C 180,E1 -20829.063,E2 -20829.063} C_VEL
LIN {X 0,Y 211.691,Z 289.963,A -85,B 0,C 180,E1 -20830.222,E2 -20830.222} C_VEL
LIN {X 0,Y 211.377,Z 293.389,A -85,B 0,C 180,E1 -20832.993,E2 -20832.993} C_VEL
LIN {X 0,Y 211.387,Z 295.542,A -85,B 0,C 180,E1 -20835.721,E2 -20835.721} C_VEL
LIN {X 0,Y 211.687,Z 296.612,A -85,B 0,C 180,E1 -20838.397,E2 -20838.397} C_VEL
LIN {X 0,Y 212.311,Z 296.668,A -85,B 0,C 180,E1 -20841.03,E2 -20841.03} C_VEL
LIN {X 0,Y 213.286,Z 295.743,A -85,B 0,C 180,E1 -20843.624,E2 -20843.624} C_VEL
LIN {X 0,Y 214.561,Z 293.851,A -85,B 0,C 180,E1 -20846.165,E2 -20846.165} C_VEL
LIN {X 0,Y 216.125,Z 290.93,A -85,B 0,C 180,E1 -20848.65,E2 -20848.65} C_VEL
LIN {X 0,Y 218.007,Z 286.866,A -85,B 0,C 180,E1 -20851.084,E2 -20851.084} C_VEL
LIN {X 0,Y 220.316,Z 281.533,A -85,B 0,C 180,E1 -20853.477,E2 -20853.477} C_VEL
LIN {X 0,Y 222.918,Z 274.83,A -85,B 0,C 180,E1 -20855.806,E2 -20855.806} C_VEL
LIN {X 0,Y 225.207,Z 268.336,A -85,B 0,C 180,E1 -20857.563,E2 -20857.563} C_VEL
LIN {X 0,Y 225.479,Z 262.123,A -85,B 0,C 180,E1 -20859.24,E2 -20859.24} C_VEL
LIN {X 0,Y 224.802,Z 254.726,A -85,B 0,C 180,E1 -20861.11,E2 -20861.11} C_VEL
LIN {X 0,Y 223.212,Z 246.43,A -85,B 0,C 180,E1 -20863.07,E2 -20863.07} C_VEL
LIN {X 0,Y 221.034,Z 238.953,A -85,B 0,C 180,E1 -20864.794,E2 -20864.794} C_VEL
LIN {X 0,Y 219.028,Z 233.295,A -85,B 0,C 180,E1 -20866.077,E2 -20866.077} C_VEL
LIN {X 0,Y 216.595,Z 228.249,A -85,B 0,C 180,E1 -20867.291,E2 -20867.291} C_VEL
LIN {X 0,Y 215.309,Z 225.168,A -85,B 0,C 180,E1 -20867.991,E2 -20867.991} C_VEL
LIN {X 0,Y 215.23,Z 224.665,A -85,B 0,C 180,E1 -20868.106,E2 -20868.106} C_VEL
LIN {X 0,Y 215.372,Z 223.273,A -85,B 0,C 180,E1 -20870.611,E2 -20870.611} C_VEL
LIN {X 0,Y 215.292,Z 221.445,A -85,B 0,C 180,E1 -20874.382,E2 -20874.382} C_VEL
LIN {X 0,Y 215.327,Z 219.83,A -85,B 0,C 180,E1 -20878.131,E2 -20878.131} C_VEL
LIN {X 0,Y 215.371,Z 219.096,A -85,B 0,C 180,E1 -20880.002,E2 -20880.002} C_VEL
LIN {X 0,Y 214.813,Z 218.01,A -85,B 0,C 180,E1 -20883.753,E2 -20883.753} C_VEL
LIN {X 0,Y 214.673,Z 217.102,A -85,B 0,C 180,E1 -20887.526,E2 -20887.526} C_VEL
LIN {X 0,Y 214.382,Z 216.529,A -85,B 0,C 180,E1 -20891.345,E2 -20891.345} C_VEL
LIN {X 0,Y 214.234,Z 216.236,A -85,B 0,C 180,E1 -20895.217,E2 -20895.217} C_VEL
LIN {X 0,Y 214.163,Z 216.275,A -85,B 0,C 180,E1 -20899.159,E2 -20899.159} C_VEL
LIN {X 0,Y 214.203,Z 216.688,A -85,B 0,C 180,E1 -20903.267,E2 -20903.267} C_VEL
LIN {X 0,Y 214.398,Z 217.574,A -85,B 0,C 180,E1 -20907.741,E2 -20907.741} C_VEL
LIN {X 0,Y 214.604,Z 218.75,A -85,B 0,C 180,E1 -20911.629,E2 -20911.629} C_VEL
LIN {X 0,Y 214.929,Z 220.531,A -85,B 0,C 180,E1 -20916.058,E2 -20916.058} C_VEL
LIN {X 0,Y 215.333,Z 222.935,A -85,B 0,C 180,E1 -20920.751,E2 -20920.751} C_VEL
LIN {X 0,Y 215.672,Z 225.063,A -85,B 0,C 180,E1 -20924.201,E2 -20924.201} C_VEL
LIN {X 0,Y 216.195,Z 227.985,A -85,B 0,C 180,E1 -20928.391,E2 -20928.391} C_VEL
LIN {X 0,Y 216.723,Z 230.791,A -85,B 0,C 180,E1 -20931.965,E2 -20931.965} C_VEL
LIN {X 0,Y 217.169,Z 233.865,A -85,B 0,C 180,E1 -20935.505,E2 -20935.505} C_VEL
LIN {X 0,Y 217.219,Z 234.911,A -85,B 0,C 180,E1 -20936.632,E2 -20936.632} C_VEL
LIN {X 0,Y 218.077,Z 238.193,A -85,B 0,C 180,E1 -20937.147,E2 -20937.147} C_VEL
LIN {X 0,Y 218.88,Z 240.365,A -85,B 0,C 180,E1 -20937.575,E2 -20937.575} C_VEL
LIN {X 0,Y 220.971,Z 248.3,A -85,B 0,C 180,E1 -20938.981,E2 -20938.981} C_VEL
LIN {X 0,Y 222.641,Z 257.246,A -85,B 0,C 180,E1 -20940.634,E2 -20940.634} C_VEL
LIN {X 0,Y 223.512,Z 265.685,A -85,B 0,C 180,E1 -20942.269,E2 -20942.269} C_VEL
LIN {X 0,Y 223.631,Z 273.472,A -85,B 0,C 180,E1 -20943.907,E2 -20943.907} C_VEL
LIN {X 0,Y 223.28,Z 279.699,A -85,B 0,C 180,E1 -20945.351,E2 -20945.351} C_VEL
LIN {X 0,Y 222.254,Z 286.622,A -85,B 0,C 180,E1 -20947.137,E2 -20947.137} C_VEL
LIN {X 0,Y 220.402,Z 292.988,A -85,B 0,C 180,E1 -20948.978,E2 -20948.978} C_VEL
LIN {X 0,Y 219.824,Z 294.488,A -85,B 0,C 180,E1 -20949.443,E2 -20949.443} C_VEL
LIN {X 0,Y 217.744,Z 297.999,A -85,B 0,C 180,E1 -20950.569,E2 -20950.569} C_VEL
LIN {X 0,Y 213.001,Z 303.097,A -85,B 0,C 180,E1 -20952.453,E2 -20952.453} C_VEL
LIN {X 0,Y 208.573,Z 307.31,A -85,B 0,C 180,E1 -20954.565,E2 -20954.565} C_VEL
LIN {X 0,Y 207.021,Z 309.376,A -85,B 0,C 180,E1 -20956.022,E2 -20956.022} C_VEL
LIN {X 0,Y 205.938,Z 311.797,A -85,B 0,C 180,E1 -20958.185,E2 -20958.185} C_VEL
LIN {X 0,Y 205.219,Z 313.433,A -85,B 0,C 180,E1 -20960.141,E2 -20960.141} C_VEL
LIN {X 0,Y 204.759,Z 314.491,A -85,B 0,C 180,E1 -20962.109,E2 -20962.109} C_VEL
LIN {X 0,Y 204.442,Z 315.175,A -85,B 0,C 180,E1 -20965.513,E2 -20965.513} C_VEL
LIN {X 0,Y 204.615,Z 314.745,A -85,B 0,C 180,E1 -20968.032,E2 -20968.032} C_VEL
LIN {X 0,Y 204.678,Z 313.849,A -85,B 0,C 180,E1 -20970,E2 -20970} C_VEL
LIN {X 0,Y 204.616,Z 311.365,A -85,B 0,C 180,E1 -20972.954,E2 -20972.954} C_VEL
LIN {X 0,Y 204.646,Z 307.545,A -85,B 0,C 180,E1 -20975.914,E2 -20975.914} C_VEL
LIN {X 0,Y 204.869,Z 304.202,A -85,B 0,C 180,E1 -20977.887,E2 -20977.887} C_VEL
LIN {X 0,Y 205.354,Z 298.946,A -85,B 0,C 180,E1 -20980.351,E2 -20980.351} C_VEL
LIN {X 0,Y 205.96,Z 293.753,A -85,B 0,C 180,E1 -20982.314,E2 -20982.314} C_VEL
LIN {X 0,Y 206.715,Z 287.474,A -85,B 0,C 180,E1 -20984.27,E2 -20984.27} C_VEL
LIN {X 0,Y 207.969,Z 278.839,A -85,B 0,C 180,E1 -20986.441,E2 -20986.441} C_VEL
LIN {X 0,Y 207.928,Z 269.681,A -85,B 0,C 180,E1 -20988.254,E2 -20988.254} C_VEL
LIN {X 0,Y 207.54,Z 261.149,A -85,B 0,C 180,E1 -20989.628,E2 -20989.628} C_VEL
LIN {X 0,Y 207.005,Z 252.486,A -85,B 0,C 180,E1 -20990.755,E2 -20990.755} C_VEL
LIN {X 0,Y 206.321,Z 243.038,A -85,B 0,C 180,E1 -20991.71,E2 -20991.71} C_VEL
LIN {X 0,Y 205.806,Z 237.074,A -85,B 0,C 180,E1 -20992.187,E2 -20992.187} C_VEL
LIN {X 0,Y 207.253,Z 229.995,A -85,B 0,C 180,E1 -20998.343,E2 -20998.343} C_VEL
LIN {X 0,Y 208.195,Z 226.41,A -85,B 0,C 180,E1 -21001.481,E2 -21001.481} C_VEL
LIN {X 0,Y 208.391,Z 223.809,A -85,B 0,C 180,E1 -21003.812,E2 -21003.812} C_VEL
LIN {X 0,Y 207.673,Z 219.916,A -85,B 0,C 180,E1 -21007.529,E2 -21007.529} C_VEL
LIN {X 0,Y 206.815,Z 215.537,A -85,B 0,C 180,E1 -21011.973,E2 -21011.973} C_VEL
LIN {X 0,Y 206.625,Z 215.555,A -85,B 0,C 180,E1 -21017.134,E2 -21017.134} C_VEL
LIN {X 0,Y 206.682,Z 215.551,A -85,B 0,C 180,E1 -21021.453,E2 -21021.453} C_VEL
LIN {X 0,Y 206.704,Z 215.545,A -85,B 0,C 180,E1 -21024.688,E2 -21024.688} C_VEL
LIN {X 0,Y 206.712,Z 215.547,A -85,B 0,C 180,E1 -21029.336,E2 -21029.336} C_VEL
LIN {X 0,Y 206.736,Z 215.543,A -85,B 0,C 180,E1 -21033.771,E2 -21033.771} C_VEL
LIN {X 0,Y 206.744,Z 215.545,A -85,B 0,C 180,E1 -21038.04,E2 -21038.04} C_VEL
LIN {X 0,Y 206.878,Z 215.525,A -85,B 0,C 180,E1 -21042.195,E2 -21042.195} C_VEL
LIN {X 0,Y 206.9,Z 215.524,A -85,B 0,C 180,E1 -21046.243,E2 -21046.243} C_VEL
LIN {X 0,Y 207.103,Z 215.495,A -85,B 0,C 180,E1 -21050.23,E2 -21050.23} C_VEL
LIN {X 0,Y 207.062,Z 215.503,A -85,B 0,C 180,E1 -21054.154,E2 -21054.154} C_VEL
LIN {X 0,Y 207.384,Z 215.459,A -85,B 0,C 180,E1 -21058.056,E2 -21058.056} C_VEL
LIN {X 0,Y 207.515,Z 215.446,A -85,B 0,C 180,E1 -21059.998,E2 -21059.998} C_VEL
LIN {X 0,Y 207.384,Z 215.463,A -85,B 0,C 180,E1 -21061.94,E2 -21061.94} C_VEL
LIN {X 0,Y 207.139,Z 215.492,A -85,B 0,C 180,E1 -21067.798,E2 -21067.798} C_VEL
LIN {X 0,Y 206.917,Z 215.521,A -85,B 0,C 180,E1 -21071.757,E2 -21071.757} C_VEL
LIN {X 0,Y 206.829,Z 215.53,A -85,B 0,C 180,E1 -21075.772,E2 -21075.772} C_VEL
LIN {X 0,Y 206.748,Z 215.543,A -85,B 0,C 180,E1 -21079.871,E2 -21079.871} C_VEL
LIN {X 0,Y 206.747,Z 215.54,A -85,B 0,C 180,E1 -21084.072,E2 -21084.072} C_VEL
LIN {X 0,Y 206.743,Z 215.546,A -85,B 0,C 180,E1 -21088.417,E2 -21088.417} C_VEL
LIN {X 0,Y 206.708,Z 215.546,A -85,B 0,C 180,E1 -21092.954,E2 -21092.954} C_VEL
LIN {X 0,Y 206.72,Z 215.546,A -85,B 0,C 180,E1 -21095.318,E2 -21095.318} C_VEL
LIN {X 0,Y 206.663,Z 215.552,A -85,B 0,C 180,E1 -21100.248,E2 -21100.248} C_VEL
LIN {X 0,Y 206.63,Z 215.559,A -85,B 0,C 180,E1 -21105.58,E2 -21105.58} C_VEL
LIN {X 0,Y 206.656,Z 215.554,A -85,B 0,C 180,E1 -21109.747,E2 -21109.747} C_VEL
LIN {X 0,Y 206.694,Z 215.548,A -85,B 0,C 180,E1 -21114.687,E2 -21114.687} C_VEL
LIN {X 0,Y 206.719,Z 215.547,A -85,B 0,C 180,E1 -21119.338,E2 -21119.338} C_VEL
LIN {X 0,Y 206.727,Z 215.544,A -85,B 0,C 180,E1 -21123.771,E2 -21123.771} C_VEL
LIN {X 0,Y 206.752,Z 215.542,A -85,B 0,C 180,E1 -21128.042,E2 -21128.042} C_VEL
LIN {X 0,Y 206.867,Z 215.526,A -85,B 0,C 180,E1 -21132.196,E2 -21132.196} C_VEL
LIN {X 0,Y 206.908,Z 215.522,A -85,B 0,C 180,E1 -21136.245,E2 -21136.245} C_VEL
LIN {X 0,Y 207.099,Z 215.498,A -85,B 0,C 180,E1 -21140.231,E2 -21140.231} C_VEL
LIN {X 0,Y 207.161,Z 215.487,A -85,B 0,C 180,E1 -21142.2,E2 -21142.2} C_VEL
LIN {X 0,Y 207.375,Z 215.464,A -85,B 0,C 180,E1 -21148.057,E2 -21148.057} C_VEL
LIN {X 0,Y 207.508,Z 215.445,A -85,B 0,C 180,E1 -21150,E2 -21150} C_VEL
LIN {X 0,Y 207.376,Z 215.463,A -85,B 0,C 180,E1 -21151.942,E2 -21151.942} C_VEL
LIN {X 0,Y 207.144,Z 215.491,A -85,B 0,C 180,E1 -21157.799,E2 -21157.799} C_VEL
LIN {X 0,Y 207.022,Z 215.507,A -85,B 0,C 180,E1 -21160.116,E2 -21160.116} C_VEL
LIN {X 0,Y 206.537,Z 215.569,A -85,B 0,C 180,E1 -21163.78,E2 -21163.78} C_VEL
LIN {X 0,Y 206.204,Z 215.797,A -85,B 0,C 180,E1 -21166.204,E2 -21166.204} C_VEL
LIN {X 0,Y 205.506,Z 220.736,A -85,B 0,C 180,E1 -21172.097,E2 -21172.097} C_VEL
LIN {X 0,Y 205.356,Z 222.171,A -85,B 0,C 180,E1 -21173.775,E2 -21173.775} C_VEL
LIN {X 0,Y 207.076,Z 232.71,A -85,B 0,C 180,E1 -21174.834,E2 -21174.834} C_VEL
LIN {X 0,Y 208.358,Z 241.777,A -85,B 0,C 180,E1 -21176.008,E2 -21176.008} C_VEL
LIN {X 0,Y 209.299,Z 249.456,A -85,B 0,C 180,E1 -21177.226,E2 -21177.226} C_VEL
LIN {X 0,Y 209.474,Z 253.968,A -85,B 0,C 180,E1 -21178.015,E2 -21178.015} C_VEL
LIN {X 0,Y 208.424,Z 261.995,A -85,B 0,C 180,E1 -21179.652,E2 -21179.652} C_VEL
LIN {X 0,Y 207.335,Z 269.765,A -85,B 0,C 180,E1 -21181.619,E2 -21181.619} C_VEL
LIN {X 0,Y 206.471,Z 276.049,A -85,B 0,C 180,E1 -21183.582,E2 -21183.582} C_VEL
LIN {X 0,Y 205.575,Z 282.582,A -85,B 0,C 180,E1 -21186.112,E2 -21186.112} C_VEL
LIN {X 0,Y 204.877,Z 287.767,A -85,B 0,C 180,E1 -21188.758,E2 -21188.758} C_VEL
LIN {X 0,Y 204.489,Z 291.014,A -85,B 0,C 180,E1 -21190.881,E2 -21190.881} C_VEL
LIN {X 0,Y 204.26,Z 294.168,A -85,B 0,C 180,E1 -21193.738,E2 -21193.738} C_VEL
LIN {X 0,Y 204.344,Z 296.146,A -85,B 0,C 180,E1 -21196.542,E2 -21196.542} C_VEL
LIN {X 0,Y 204.762,Z 297.059,A -85,B 0,C 180,E1 -21199.3,E2 -21199.3} C_VEL
LIN {X 0,Y 205.528,Z 296.963,A -85,B 0,C 180,E1 -21202.014,E2 -21202.014} C_VEL
LIN {X 0,Y 206.66,Z 295.858,A -85,B 0,C 180,E1 -21204.704,E2 -21204.704} C_VEL
LIN {X 0,Y 208.218,Z 293.484,A -85,B 0,C 180,E1 -21207.546,E2 -21207.546} C_VEL
LIN {X 0,Y 210.255,Z 289.855,A -85,B 0,C 180,E1 -21210.351,E2 -21210.351} C_VEL
LIN {X 0,Y 211.993,Z 286.382,A -85,B 0,C 180,E1 -21212.348,E2 -21212.348} C_VEL
LIN {X 0,Y 214.5,Z 280.886,A -85,B 0,C 180,E1 -21214.792,E2 -21214.792} C_VEL
LIN {X 0,Y 217.361,Z 273.861,A -85,B 0,C 180,E1 -21217.172,E2 -21217.172} C_VEL
LIN {X 0,Y 218.999,Z 268.916,A -85,B 0,C 180,E1 -21218.536,E2 -21218.536} C_VEL
LIN {X 0,Y 219.096,Z 261.704,A -85,B 0,C 180,E1 -21220.599,E2 -21220.599} C_VEL
LIN {X 0,Y 218.25,Z 253.927,A -85,B 0,C 180,E1 -21222.673,E2 -21222.673} C_VEL
LIN {X 0,Y 216.785,Z 246.756,A -85,B 0,C 180,E1 -21224.489,E2 -21224.489} C_VEL
LIN {X 0,Y 214.048,Z 237.78,A -85,B 0,C 180,E1 -21226.714,E2 -21226.714} C_VEL
LIN {X 0,Y 211.609,Z 232.269,A -85,B 0,C 180,E1 -21228.199,E2 -21228.199} C_VEL
LIN {X 0,Y 210.13,Z 228.954,A -85,B 0,C 180,E1 -21229.036,E2 -21229.036} C_VEL
LIN {X 0,Y 208.677,Z 226.171,A -85,B 0,C 180,E1 -21229.818,E2 -21229.818} C_VEL
LIN {X 0,Y 208.419,Z 225.096,A -85,B 0,C 180,E1 -21230.05,E2 -21230.05} C_VEL
LIN {X 0,Y 208.395,Z 223.125,A -85,B 0,C 180,E1 -21234.195,E2 -21234.195} C_VEL
LIN {X 0,Y 208.429,Z 221.521,A -85,B 0,C 180,E1 -21238.069,E2 -21238.069} C_VEL
LIN {X 0,Y 208.484,Z 220.799,A -85,B 0,C 180,E1 -21240.002,E2 -21240.002} C_VEL
LIN {X 0,Y 207.944,Z 219.738,A -85,B 0,C 180,E1 -21243.877,E2 -21243.877} C_VEL
LIN {X 0,Y 207.804,Z 218.865,A -85,B 0,C 180,E1 -21247.776,E2 -21247.776} C_VEL
LIN {X 0,Y 207.495,Z 218.347,A -85,B 0,C 180,E1 -21251.727,E2 -21251.727} C_VEL
LIN {X 0,Y 207.378,Z 218.117,A -85,B 0,C 180,E1 -21255.732,E2 -21255.732} C_VEL
LIN {X 0,Y 207.314,Z 218.237,A -85,B 0,C 180,E1 -21259.818,E2 -21259.818} C_VEL
LIN {X 0,Y 207.364,Z 218.731,A -85,B 0,C 180,E1 -21264,E2 -21264} C_VEL
LIN {X 0,Y 207.574,Z 219.635,A -85,B 0,C 180,E1 -21268.321,E2 -21268.321} C_VEL
LIN {X 0,Y 207.788,Z 221.035,A -85,B 0,C 180,E1 -21272.765,E2 -21272.765} C_VEL
LIN {X 0,Y 208.052,Z 222.258,A -85,B 0,C 180,E1 -21275.834,E2 -21275.834} C_VEL
LIN {X 0,Y 208.354,Z 224.229,A -85,B 0,C 180,E1 -21279.86,E2 -21279.86} C_VEL
LIN {X 0,Y 208.572,Z 225.625,A -85,B 0,C 180,E1 -21282.372,E2 -21282.372} C_VEL
LIN {X 0,Y 208.849,Z 227.286,A -85,B 0,C 180,E1 -21285.035,E2 -21285.035} C_VEL
LIN {X 0,Y 209.186,Z 229.14,A -85,B 0,C 180,E1 -21287.784,E2 -21287.784} C_VEL
LIN {X 0,Y 209.57,Z 231.128,A -85,B 0,C 180,E1 -21290.474,E2 -21290.474} C_VEL
LIN {X 0,Y 210.164,Z 234.701,A -85,B 0,C 180,E1 -21294.686,E2 -21294.686} C_VEL
LIN {X 0,Y 211.382,Z 237.916,A -85,B 0,C 180,E1 -21295.349,E2 -21295.349} C_VEL
LIN {X 0,Y 212.452,Z 239.943,A -85,B 0,C 180,E1 -21295.885,E2 -21295.885} C_VEL
LIN {X 0,Y 214.554,Z 246.868,A -85,B 0,C 180,E1 -21297.268,E2 -21297.268} C_VEL
LIN {X 0,Y 216.406,Z 256.726,A -85,B 0,C 180,E1 -21299.199,E2 -21299.199} C_VEL
LIN {X 0,Y 217.283,Z 265.287,A -85,B 0,C 180,E1 -21300.976,E2 -21300.976} C_VEL
LIN {X 0,Y 217.365,Z 273.428,A -85,B 0,C 180,E1 -21302.775,E2 -21302.775} C_VEL
LIN {X 0,Y 216.89,Z 280.756,A -85,B 0,C 180,E1 -21304.574,E2 -21304.574} C_VEL
LIN {X 0,Y 215.732,Z 287.518,A -85,B 0,C 180,E1 -21306.425,E2 -21306.425} C_VEL
LIN {X 0,Y 213.827,Z 293.588,A -85,B 0,C 180,E1 -21308.299,E2 -21308.299} C_VEL
LIN {X 0,Y 211.249,Z 299.721,A -85,B 0,C 180,E1 -21310.568,E2 -21310.568} C_VEL
LIN {X 0,Y 208.757,Z 305.427,A -85,B 0,C 180,E1 -21313.372,E2 -21313.372} C_VEL
LIN {X 0,Y 207.021,Z 309.376,A -85,B 0,C 180,E1 -21316.022,E2 -21316.022} C_VEL
LIN {X 0,Y 205.562,Z 311.244,A -85,B 0,C 180,E1 -21317.537,E2 -21317.537} C_VEL
LIN {X 0,Y 201.713,Z 313.385,A -85,B 0,C 180,E1 -21320.036,E2 -21320.036} C_VEL
LIN {X 0,Y 198.235,Z 314.565,A -85,B 0,C 180,E1 -21322.674,E2 -21322.674} C_VEL
LIN {X 0,Y 197.383,Z 314.749,A -85,B 0,C 180,E1 -21324.366,E2 -21324.366} C_VEL
LIN {X 0,Y 197.543,Z 314.254,A -85,B 0,C 180,E1 -21327.962,E2 -21327.962} C_VEL
LIN {X 0,Y 197.613,Z 313.287,A -85,B 0,C 180,E1 -21330,E2 -21330} C_VEL
LIN {X 0,Y 197.611,Z 311.737,A -85,B 0,C 180,E1 -21332.039,E2 -21332.039} C_VEL
LIN {X 0,Y 197.576,Z 308.225,A -85,B 0,C 180,E1 -21335.118,E2 -21335.118} C_VEL
LIN {X 0,Y 197.682,Z 305.175,A -85,B 0,C 180,E1 -21337.148,E2 -21337.148} C_VEL
LIN {X 0,Y 198.143,Z 300.242,A -85,B 0,C 180,E1 -21339.7,E2 -21339.7} C_VEL
LIN {X 0,Y 198.601,Z 295.379,A -85,B 0,C 180,E1 -21341.741,E2 -21341.741} C_VEL
LIN {X 0,Y 199.382,Z 289.512,A -85,B 0,C 180,E1 -21343.765,E2 -21343.765} C_VEL
LIN {X 0,Y 200.284,Z 282.327,A -85,B 0,C 180,E1 -21345.781,E2 -21345.781} C_VEL
LIN {X 0,Y 201.04,Z 277.097,A -85,B 0,C 180,E1 -21347.025,E2 -21347.025} C_VEL
LIN {X 0,Y 200.794,Z 268.517,A -85,B 0,C 180,E1 -21348.745,E2 -21348.745} C_VEL
LIN {X 0,Y 200.487,Z 260.358,A -85,B 0,C 180,E1 -21350.082,E2 -21350.082} C_VEL
LIN {X 0,Y 199.927,Z 251.51,A -85,B 0,C 180,E1 -21351.255,E2 -21351.255} C_VEL
LIN {X 0,Y 199.103,Z 240.883,A -85,B 0,C 180,E1 -21352.335,E2 -21352.335} C_VEL
LIN {X 0,Y 198.778,Z 236.795,A -85,B 0,C 180,E1 -21352.682,E2 -21352.682} C_VEL
LIN {X 0,Y 200.224,Z 230.178,A -85,B 0,C 180,E1 -21358.653,E2 -21358.653} C_VEL
LIN {X 0,Y 201.119,Z 226.905,A -85,B 0,C 180,E1 -21361.613,E2 -21361.613} C_VEL
LIN {X 0,Y 201.318,Z 224.414,A -85,B 0,C 180,E1 -21363.957,E2 -21363.957} C_VEL
LIN {X 0,Y 200.552,Z 220.505,A -85,B 0,C 180,E1 -21367.826,E2 -21367.826} C_VEL
LIN {X 0,Y 199.767,Z 216.415,A -85,B 0,C 180,E1 -21372.204,E2 -21372.204} C_VEL
LIN {X 0,Y 199.579,Z 216.434,A -85,B 0,C 180,E1 -21378.003,E2 -21378.003} C_VEL
LIN {X 0,Y 199.605,Z 216.433,A -85,B 0,C 180,E1 -21380.77,E2 -21380.77} C_VEL
LIN {X 0,Y 199.617,Z 216.428,A -85,B 0,C 180,E1 -21385.713,E2 -21385.713} C_VEL
LIN {X 0,Y 199.698,Z 216.424,A -85,B 0,C 180,E1 -21388.135,E2 -21388.135} C_VEL
LIN {X 0,Y 199.689,Z 216.418,A -85,B 0,C 180,E1 -21392.771,E2 -21392.771} C_VEL
LIN {X 0,Y 199.719,Z 216.419,A -85,B 0,C 180,E1 -21397.225,E2 -21397.225} C_VEL
LIN {X 0,Y 199.801,Z 216.407,A -85,B 0,C 180,E1 -21401.757,E2 -21401.757} C_VEL
LIN {X 0,Y 199.84,Z 216.405,A -85,B 0,C 180,E1 -21405.747,E2 -21405.747} C_VEL
LIN {X 0,Y 200.026,Z 216.378,A -85,B 0,C 180,E1 -21409.88,E2 -21409.88} C_VEL
LIN {X 0,Y 200.023,Z 216.381,A -85,B 0,C 180,E1 -21413.948,E2 -21413.948} C_VEL
LIN {X 0,Y 200.324,Z 216.339,A -85,B 0,C 180,E1 -21417.988,E2 -21417.988} C_VEL
LIN {X 0,Y 200.479,Z 216.322,A -85,B 0,C 180,E1 -21419.998,E2 -21419.998} C_VEL
LIN {X 0,Y 200.028,Z 216.379,A -85,B 0,C 180,E1 -21424.028,E2 -21424.028} C_VEL
LIN {X 0,Y 200.088,Z 216.37,A -85,B 0,C 180,E1 -21428.075,E2 -21428.075} C_VEL
LIN {X 0,Y 199.866,Z 216.4,A -85,B 0,C 180,E1 -21432.178,E2 -21432.178} C_VEL
LIN {X 0,Y 199.766,Z 216.411,A -85,B 0,C 180,E1 -21436.345,E2 -21436.345} C_VEL
LIN {X 0,Y 199.672,Z 216.426,A -85,B 0,C 180,E1 -21440.606,E2 -21440.606} C_VEL
LIN {X 0,Y 199.664,Z 216.425,A -85,B 0,C 180,E1 -21444.983,E2 -21444.983} C_VEL
LIN {X 0,Y 199.674,Z 216.423,A -85,B 0,C 180,E1 -21449.52,E2 -21449.52} C_VEL
LIN {X 0,Y 199.663,Z 216.424,A -85,B 0,C 180,E1 -21452.35,E2 -21452.35} C_VEL
LIN {X 0,Y 199.638,Z 216.428,A -85,B 0,C 180,E1 -21456.757,E2 -21456.757} C_VEL
LIN {X 0,Y 199.636,Z 216.426,A -85,B 0,C 180,E1 -21459.319,E2 -21459.319} C_VEL
LIN {X 0,Y 199.577,Z 216.436,A -85,B 0,C 180,E1 -21464.769,E2 -21464.769} C_VEL
LIN {X 0,Y 199.575,Z 216.435,A -85,B 0,C 180,E1 -21468.003,E2 -21468.003} C_VEL
LIN {X 0,Y 199.606,Z 216.431,A -85,B 0,C 180,E1 -21470.766,E2 -21470.766} C_VEL
LIN {X 0,Y 199.61,Z 216.431,A -85,B 0,C 180,E1 -21475.712,E2 -21475.712} C_VEL
LIN {X 0,Y 199.697,Z 216.42,A -85,B 0,C 180,E1 -21478.136,E2 -21478.136} C_VEL
LIN {X 0,Y 199.682,Z 216.422,A -85,B 0,C 180,E1 -21482.77,E2 -21482.77} C_VEL
LIN {X 0,Y 199.732,Z 216.417,A -85,B 0,C 180,E1 -21487.228,E2 -21487.228} C_VEL
LIN {X 0,Y 199.79,Z 216.408,A -85,B 0,C 180,E1 -21491.757,E2 -21491.757} C_VEL
LIN {X 0,Y 199.842,Z 216.403,A -85,B 0,C 180,E1 -21495.748,E2 -21495.748} C_VEL
LIN {X 0,Y 200.064,Z 216.374,A -85,B 0,C 180,E1 -21499.883,E2 -21499.883} C_VEL
LIN {X 0,Y 200.028,Z 216.378,A -85,B 0,C 180,E1 -21503.949,E2 -21503.949} C_VEL
LIN {X 0,Y 200.315,Z 216.343,A -85,B 0,C 180,E1 -21507.989,E2 -21507.989} C_VEL
LIN {X 0,Y 200.472,Z 216.321,A -85,B 0,C 180,E1 -21510,E2 -21510} C_VEL
LIN {X 0,Y 200.025,Z 216.38,A -85,B 0,C 180,E1 -21514.029,E2 -21514.029} C_VEL
LIN {X 0,Y 200.086,Z 216.371,A -85,B 0,C 180,E1 -21518.076,E2 -21518.076} C_VEL
LIN {X 0,Y 199.951,Z 216.389,A -85,B 0,C 180,E1 -21520.225,E2 -21520.225} C_VEL
LIN {X 0,Y 199.208,Z 216.482,A -85,B 0,C 180,E1 -21525.867,E2 -21525.867} C_VEL
LIN {X 0,Y 198.496,Z 220.281,A -85,B 0,C 180,E1 -21530.736,E2 -21530.736} C_VEL
LIN {X 0,Y 198.322,Z 222.373,A -85,B 0,C 180,E1 -21533.287,E2 -21533.287} C_VEL
LIN {X 0,Y 200.268,Z 234.664,A -85,B 0,C 180,E1 -21534.628,E2 -21534.628} C_VEL
LIN {X 0,Y 201.483,Z 243.479,A -85,B 0,C 180,E1 -21535.85,E2 -21535.85} C_VEL
LIN {X 0,Y 202.483,Z 252.456,A -85,B 0,C 180,E1 -21537.38,E2 -21537.38} C_VEL
LIN {X 0,Y 201.707,Z 260.15,A -85,B 0,C 180,E1 -21538.91,E2 -21538.91} C_VEL
LIN {X 0,Y 200.405,Z 269.04,A -85,B 0,C 180,E1 -21541.148,E2 -21541.148} C_VEL
LIN {X 0,Y 199.422,Z 275.953,A -85,B 0,C 180,E1 -21543.34,E2 -21543.34} C_VEL
LIN {X 0,Y 198.641,Z 281.573,A -85,B 0,C 180,E1 -21545.54,E2 -21545.54} C_VEL
LIN {X 0,Y 197.808,Z 287.696,A -85,B 0,C 180,E1 -21548.592,E2 -21548.592} C_VEL
LIN {X 0,Y 197.284,Z 291.967,A -85,B 0,C 180,E1 -21551.577,E2 -21551.577} C_VEL
LIN {X 0,Y 197.14,Z 294.939,A -85,B 0,C 180,E1 -21554.524,E2 -21554.524} C_VEL
LIN {X 0,Y 197.329,Z 296.751,A -85,B 0,C 180,E1 -21557.417,E2 -21557.417} C_VEL
LIN {X 0,Y 197.875,Z 297.503,A -85,B 0,C 180,E1 -21560.262,E2 -21560.262} C_VEL
LIN {X 0,Y 198.794,Z 297.217,A -85,B 0,C 180,E1 -21563.061,E2 -21563.061} C_VEL
LIN {X 0,Y 200.11,Z 295.918,A -85,B 0,C 180,E1 -21565.813,E2 -21565.813} C_VEL
LIN {X 0,Y 201.69,Z 293.658,A -85,B 0,C 180,E1 -21568.49,E2 -21568.49} C_VEL
LIN {X 0,Y 203.654,Z 290.371,A -85,B 0,C 180,E1 -21571.112,E2 -21571.112} C_VEL
LIN {X 0,Y 206.068,Z 285.926,A -85,B 0,C 180,E1 -21573.683,E2 -21573.683} C_VEL
LIN {X 0,Y 208.734,Z 280.277,A -85,B 0,C 180,E1 -21576.171,E2 -21576.171} C_VEL
LIN {X 0,Y 211.872,Z 272.817,A -85,B 0,C 180,E1 -21578.602,E2 -21578.602} C_VEL
LIN {X 0,Y 212.605,Z 270.756,A -85,B 0,C 180,E1 -21579.187,E2 -21579.187} C_VEL
LIN {X 0,Y 212.904,Z 264.209,A -85,B 0,C 180,E1 -21581.227,E2 -21581.227} C_VEL
LIN {X 0,Y 212.149,Z 255.509,A -85,B 0,C 180,E1 -21583.746,E2 -21583.746} C_VEL
LIN {X 0,Y 210.465,Z 247.309,A -85,B 0,C 180,E1 -21585.991,E2 -21585.991} C_VEL
LIN {X 0,Y 208.544,Z 240.835,A -85,B 0,C 180,E1 -21587.771,E2 -21587.771} C_VEL
LIN {X 0,Y 205.033,Z 232.76,A -85,B 0,C 180,E1 -21590.133,E2 -21590.133} C_VEL
LIN {X 0,Y 203.716,Z 230.019,A -85,B 0,C 180,E1 -21590.946,E2 -21590.946} C_VEL
LIN {X 0,Y 201.998,Z 227.184,A -85,B 0,C 180,E1 -21591.939,E2 -21591.939} C_VEL
LIN {X 0,Y 201.532,Z 225.532,A -85,B 0,C 180,E1 -21592.362,E2 -21592.362} C_VEL
LIN {X 0,Y 201.528,Z 223.23,A -85,B 0,C 180,E1 -21598.003,E2 -21598.003} C_VEL
LIN {X 0,Y 201.591,Z 222.53,A -85,B 0,C 180,E1 -21600.002,E2 -21600.002} C_VEL
LIN {X 0,Y 201.056,Z 221.486,A -85,B 0,C 180,E1 -21604.011,E2 -21604.011} C_VEL
LIN {X 0,Y 200.923,Z 220.645,A -85,B 0,C 180,E1 -21608.045,E2 -21608.045} C_VEL
LIN {X 0,Y 200.614,Z 220.18,A -85,B 0,C 180,E1 -21612.135,E2 -21612.135} C_VEL
LIN {X 0,Y 200.526,Z 220.004,A -85,B 0,C 180,E1 -21616.285,E2 -21616.285} C_VEL
LIN {X 0,Y 200.457,Z 220.205,A -85,B 0,C 180,E1 -21620.526,E2 -21620.526} C_VEL
LIN {X 0,Y 200.532,Z 220.791,A -85,B 0,C 180,E1 -21624.872,E2 -21624.872} C_VEL
LIN {X 0,Y 200.748,Z 221.812,A -85,B 0,C 180,E1 -21629.351,E2 -21629.351} C_VEL
LIN {X 0,Y 201.022,Z 223.358,A -85,B 0,C 180,E1 -21634.015,E2 -21634.015} C_VEL
LIN {X 0,Y 201.213,Z 224.422,A -85,B 0,C 180,E1 -21636.55,E2 -21636.55} C_VEL
LIN {X 0,Y 201.594,Z 226.867,A -85,B 0,C 180,E1 -21641.483,E2 -21641.483} C_VEL
LIN {X 0,Y 202,Z 229.526,A -85,B 0,C 180,E1 -21645.906,E2 -21645.906} C_VEL
LIN {X 0,Y 202.51,Z 232.155,A -85,B 0,C 180,E1 -21649.775,E2 -21649.775} C_VEL
LIN {X 0,Y 202.911,Z 234.251,A -85,B 0,C 180,E1 -21652.373,E2 -21652.373} C_VEL
LIN {X 0,Y 204.251,Z 237.543,A -85,B 0,C 180,E1 -21653.18,E2 -21653.18} C_VEL
LIN {X 0,Y 205.769,Z 240.001,A -85,B 0,C 180,E1 -21653.959,E2 -21653.959} C_VEL
LIN {X 0,Y 208.003,Z 245.683,A -85,B 0,C 180,E1 -21655.34,E2 -21655.34} C_VEL
LIN {X 0,Y 209.709,Z 252.846,A -85,B 0,C 180,E1 -21656.913,E2 -21656.913} C_VEL
LIN {X 0,Y 210.978,Z 262.517,A -85,B 0,C 180,E1 -21659.007,E2 -21659.007} C_VEL
LIN {X 0,Y 211.27,Z 272.031,A -85,B 0,C 180,E1 -21661.223,E2 -21661.223} C_VEL
LIN {X 0,Y 210.743,Z 279.931,A -85,B 0,C 180,E1 -21663.243,E2 -21663.243} C_VEL
LIN {X 0,Y 209.656,Z 286.615,A -85,B 0,C 180,E1 -21665.134,E2 -21665.134} C_VEL
LIN {X 0,Y 208.322,Z 291.451,A -85,B 0,C 180,E1 -21666.647,E2 -21666.647} C_VEL
LIN {X 0,Y 206.063,Z 296.718,A -85,B 0,C 180,E1 -21668.492,E2 -21668.492} C_VEL
LIN {X 0,Y 203.634,Z 302.094,A -85,B 0,C 180,E1 -21670.861,E2 -21670.861} C_VEL
LIN {X 0,Y 201.965,Z 305.612,A -85,B 0,C 180,E1 -21672.796,E2 -21672.796} C_VEL
LIN {X 0,Y 200.011,Z 309.694,A -85,B 0,C 180,E1 -21675.761,E2 -21675.761} C_VEL
LIN {X 0,Y 198.989,Z 311.721,A -85,B 0,C 180,E1 -21677.766,E2 -21677.766} C_VEL
LIN {X 0,Y 198.218,Z 313.259,A -85,B 0,C 180,E1 -21679.789,E2 -21679.789} C_VEL
LIN {X 0,Y 197.713,Z 314.293,A -85,B 0,C 180,E1 -21681.826,E2 -21681.826} C_VEL
LIN {X 0,Y 197.383,Z 314.749,A -85,B 0,C 180,E1 -21684.366,E2 -21684.366} C_VEL
LIN {X 0,Y 196.661,Z 314.696,A -85,B 0,C 180,E1 -21686.072,E2 -21686.072} C_VEL
LIN {X 0,Y 195.11,Z 314.189,A -85,B 0,C 180,E1 -21687.747,E2 -21687.747} C_VEL
LIN {X 0,Y 192.636,Z 312.89,A -85,B 0,C 180,E1 -21689.967,E2 -21689.967} C_VEL
LIN {X 0,Y 190.649,Z 310.688,A -85,B 0,C 180,E1 -21692.517,E2 -21692.517} C_VEL
LIN {X 0,Y 190.468,Z 309.739,A -85,B 0,C 180,E1 -21693.379,E2 -21693.379} C_VEL
LIN {X 0,Y 190.519,Z 305.908,A -85,B 0,C 180,E1 -21696.354,E2 -21696.354} C_VEL
LIN {X 0,Y 191,Z 300.291,A -85,B 0,C 180,E1 -21699.531,E2 -21699.531} C_VEL
LIN {X 0,Y 191.658,Z 294.108,A -85,B 0,C 180,E1 -21702.173,E2 -21702.173} C_VEL
LIN {X 0,Y 192.438,Z 288.043,A -85,B 0,C 180,E1 -21704.272,E2 -21704.272} C_VEL
LIN {X 0,Y 193.307,Z 281.664,A -85,B 0,C 180,E1 -21706.095,E2 -21706.095} C_VEL
LIN {X 0,Y 193.968,Z 276.34,A -85,B 0,C 180,E1 -21707.393,E2 -21707.393} C_VEL
LIN {X 0,Y 193.72,Z 268.315,A -85,B 0,C 180,E1 -21709.058,E2 -21709.058} C_VEL
LIN {X 0,Y 193.42,Z 259.963,A -85,B 0,C 180,E1 -21710.477,E2 -21710.477} C_VEL
LIN {X 0,Y 192.897,Z 251.479,A -85,B 0,C 180,E1 -21711.648,E2 -21711.648} C_VEL
LIN {X 0,Y 192.138,Z 240.984,A -85,B 0,C 180,E1 -21712.764,E2 -21712.764} C_VEL
LIN {X 0,Y 191.783,Z 236.513,A -85,B 0,C 180,E1 -21713.2,E2 -21713.2} C_VEL
LIN {X 0,Y 192.99,Z 231.132,A -85,B 0,C 180,E1 -21718.257,E2 -21718.257} C_VEL
LIN {X 0,Y 194.045,Z 227.499,A -85,B 0,C 180,E1 -21721.68,E2 -21721.68} C_VEL
LIN {X 0,Y 194.266,Z 225.418,A -85,B 0,C 180,E1 -21723.685,E2 -21723.685} C_VEL
LIN {X 0,Y 193.426,Z 221.068,A -85,B 0,C 180,E1 -21728.148,E2 -21728.148} C_VEL
LIN {X 0,Y 192.739,Z 217.29,A -85,B 0,C 180,E1 -21732.246,E2 -21732.246} C_VEL
LIN {X 0,Y 192.517,Z 217.313,A -85,B 0,C 180,E1 -21736.897,E2 -21736.897} C_VEL
LIN {X 0,Y 192.549,Z 217.312,A -85,B 0,C 180,E1 -21741.646,E2 -21741.646} C_VEL
LIN {X 0,Y 192.601,Z 217.304,A -85,B 0,C 180,E1 -21746.813,E2 -21746.813} C_VEL
LIN {X 0,Y 192.665,Z 217.298,A -85,B 0,C 180,E1 -21751.69,E2 -21751.69} C_VEL
LIN {X 0,Y 192.69,Z 217.294,A -85,B 0,C 180,E1 -21756.345,E2 -21756.345} C_VEL
LIN {X 0,Y 192.736,Z 217.287,A -85,B 0,C 180,E1 -21761.457,E2 -21761.457} C_VEL
LIN {X 0,Y 192.768,Z 217.285,A -85,B 0,C 180,E1 -21765.212,E2 -21765.212} C_VEL
LIN {X 0,Y 192.949,Z 217.26,A -85,B 0,C 180,E1 -21769.565,E2 -21769.565} C_VEL
LIN {X 0,Y 192.986,Z 217.258,A -85,B 0,C 180,E1 -21773.726,E2 -21773.726} C_VEL
LIN {X 0,Y 193.265,Z 217.218,A -85,B 0,C 180,E1 -21777.914,E2 -21777.914} C_VEL
LIN {X 0,Y 193.444,Z 217.199,A -85,B 0,C 180,E1 -21779.998,E2 -21779.998} C_VEL
LIN {X 0,Y 192.974,Z 217.258,A -85,B 0,C 180,E1 -21784.175,E2 -21784.175} C_VEL
LIN {X 0,Y 193.036,Z 217.249,A -85,B 0,C 180,E1 -21788.372,E2 -21788.372} C_VEL
LIN {X 0,Y 192.793,Z 217.283,A -85,B 0,C 180,E1 -21792.632,E2 -21792.632} C_VEL
LIN {X 0,Y 192.719,Z 217.292,A -85,B 0,C 180,E1 -21796.96,E2 -21796.96} C_VEL
LIN {X 0,Y 192.609,Z 217.302,A -85,B 0,C 180,E1 -21801.398,E2 -21801.398} C_VEL
LIN {X 0,Y 192.647,Z 217.296,A -85,B 0,C 180,E1 -21804.211,E2 -21804.211} C_VEL
LIN {X 0,Y 192.649,Z 217.299,A -85,B 0,C 180,E1 -21808.89,E2 -21808.89} C_VEL
LIN {X 0,Y 192.599,Z 217.303,A -85,B 0,C 180,E1 -21813.183,E2 -21813.183} C_VEL
LIN {X 0,Y 192.607,Z 217.305,A -85,B 0,C 180,E1 -21816.605,E2 -21816.605} C_VEL
LIN {X 0,Y 192.521,Z 217.312,A -85,B 0,C 180,E1 -21821.076,E2 -21821.076} C_VEL
LIN {X 0,Y 192.488,Z 217.32,A -85,B 0,C 180,E1 -21826.074,E2 -21826.074} C_VEL
LIN {X 0,Y 192.514,Z 217.317,A -85,B 0,C 180,E1 -21830.049,E2 -21830.049} C_VEL
LIN {X 0,Y 192.556,Z 217.31,A -85,B 0,C 180,E1 -21834.269,E2 -21834.269} C_VEL
LIN {X 0,Y 192.606,Z 217.3,A -85,B 0,C 180,E1 -21837.056,E2 -21837.056} C_VEL
LIN {X 0,Y 192.66,Z 217.299,A -85,B 0,C 180,E1 -21841.691,E2 -21841.691} C_VEL
LIN {X 0,Y 192.7,Z 217.29,A -85,B 0,C 180,E1 -21846.347,E2 -21846.347} C_VEL
LIN {X 0,Y 192.726,Z 217.289,A -85,B 0,C 180,E1 -21851.456,E2 -21851.456} C_VEL
LIN {X 0,Y 192.766,Z 217.285,A -85,B 0,C 180,E1 -21855.213,E2 -21855.213} C_VEL
LIN {X 0,Y 192.975,Z 217.258,A -85,B 0,C 180,E1 -21859.508,E2 -21859.508} C_VEL
LIN {X 0,Y 193.055,Z 217.244,A -85,B 0,C 180,E1 -21861.627,E2 -21861.627} C_VEL
LIN {X 0,Y 193.257,Z 217.222,A -85,B 0,C 180,E1 -21867.916,E2 -21867.916} C_VEL
LIN {X 0,Y 193.436,Z 217.197,A -85,B 0,C 180,E1 -21870,E2 -21870} C_VEL
LIN {X 0,Y 192.971,Z 217.26,A -85,B 0,C 180,E1 -21874.177,E2 -21874.177} C_VEL
LIN {X 0,Y 193.026,Z 217.251,A -85,B 0,C 180,E1 -21878.374,E2 -21878.374} C_VEL
LIN {X 0,Y 192.847,Z 217.275,A -85,B 0,C 180,E1 -21880.499,E2 -21880.499} C_VEL
LIN {X 0,Y 192.108,Z 217.367,A -85,B 0,C 180,E1 -21886.061,E2 -21886.061} C_VEL
LIN {X 0,Y 191.316,Z 222.679,A -85,B 0,C 180,E1 -21892.822,E2 -21892.822} C_VEL
LIN {X 0,Y 193.192,Z 234.694,A -85,B 0,C 180,E1 -21894.158,E2 -21894.158} C_VEL
LIN {X 0,Y 194.429,Z 243.672,A -85,B 0,C 180,E1 -21895.448,E2 -21895.448} C_VEL
LIN {X 0,Y 195.431,Z 252.467,A -85,B 0,C 180,E1 -21897.001,E2 -21897.001} C_VEL
LIN {X 0,Y 195.127,Z 257.035,A -85,B 0,C 180,E1 -21897.919,E2 -21897.919} C_VEL
LIN {X 0,Y 194.052,Z 264.503,A -85,B 0,C 180,E1 -21899.638,E2 -21899.638} C_VEL
LIN {X 0,Y 192.922,Z 272.401,A -85,B 0,C 180,E1 -21901.885,E2 -21901.885} C_VEL
LIN {X 0,Y 191.848,Z 279.809,A -85,B 0,C 180,E1 -21904.598,E2 -21904.598} C_VEL
LIN {X 0,Y 191.171,Z 284.381,A -85,B 0,C 180,E1 -21906.682,E2 -21906.682} C_VEL
LIN {X 0,Y 190.566,Z 288.87,A -85,B 0,C 180,E1 -21909.246,E2 -21909.246} C_VEL
LIN {X 0,Y 190.113,Z 292.919,A -85,B 0,C 180,E1 -21912.327,E2 -21912.327} C_VEL
LIN {X 0,Y 190.061,Z 295.696,A -85,B 0,C 180,E1 -21915.369,E2 -21915.369} C_VEL
LIN {X 0,Y 190.363,Z 297.326,A -85,B 0,C 180,E1 -21918.356,E2 -21918.356} C_VEL
LIN {X 0,Y 191.043,Z 297.87,A -85,B 0,C 180,E1 -21921.292,E2 -21921.292} C_VEL
LIN {X 0,Y 192.136,Z 297.394,A -85,B 0,C 180,E1 -21924.182,E2 -21924.182} C_VEL
LIN {X 0,Y 193.615,Z 295.948,A -85,B 0,C 180,E1 -21927.013,E2 -21927.013} C_VEL
LIN {X 0,Y 195.421,Z 293.538,A -85,B 0,C 180,E1 -21929.771,E2 -21929.771} C_VEL
LIN {X 0,Y 197.58,Z 290.112,A -85,B 0,C 180,E1 -21932.459,E2 -21932.459} C_VEL
LIN {X 0,Y 200.708,Z 284.584,A -85,B 0,C 180,E1 -21935.562,E2 -21935.562} C_VEL
LIN {X 0,Y 203.743,Z 278.281,A -85,B 0,C 180,E1 -21938.098,E2 -21938.098} C_VEL
LIN {X 0,Y 205.959,Z 273.355,A -85,B 0,C 180,E1 -21939.682,E2 -21939.682} C_VEL
LIN {X 0,Y 206.522,Z 270.508,A -85,B 0,C 180,E1 -21940.624,E2 -21940.624} C_VEL
LIN {X 0,Y 206.583,Z 262.642,A -85,B 0,C 180,E1 -21943.194,E2 -21943.194} C_VEL
LIN {X 0,Y 205.691,Z 254.499,A -85,B 0,C 180,E1 -21945.659,E2 -21945.659} C_VEL
LIN {X 0,Y 204.348,Z 248.312,A -85,B 0,C 180,E1 -21947.516,E2 -21947.516} C_VEL
LIN {X 0,Y 201.731,Z 240.295,A -85,B 0,C 180,E1 -21949.97,E2 -21949.97} C_VEL
LIN {X 0,Y 199.902,Z 235.854,A -85,B 0,C 180,E1 -21951.409,E2 -21951.409} C_VEL
LIN {X 0,Y 197.809,Z 232.157,A -85,B 0,C 180,E1 -21952.756,E2 -21952.756} C_VEL
LIN {X 0,Y 197.234,Z 230.903,A -85,B 0,C 180,E1 -21953.159,E2 -21953.159} C_VEL
LIN {X 0,Y 195.126,Z 227.812,A -85,B 0,C 180,E1 -21954.512,E2 -21954.512} C_VEL
LIN {X 0,Y 194.537,Z 226.031,A -85,B 0,C 180,E1 -21955.08,E2 -21955.08} C_VEL
LIN {X 0,Y 194.714,Z 224.264,A -85,B 0,C 180,E1 -21960.002,E2 -21960.002} C_VEL
LIN {X 0,Y 194.179,Z 223.254,A -85,B 0,C 180,E1 -21964.153,E2 -21964.153} C_VEL
LIN {X 0,Y 194.047,Z 222.449,A -85,B 0,C 180,E1 -21968.332,E2 -21968.332} C_VEL
LIN {X 0,Y 193.741,Z 222.032,A -85,B 0,C 180,E1 -21972.573,E2 -21972.573} C_VEL
LIN {X 0,Y 193.657,Z 221.919,A -85,B 0,C 180,E1 -21976.879,E2 -21976.879} C_VEL
LIN {X 0,Y 193.603,Z 222.202,A -85,B 0,C 180,E1 -21981.287,E2 -21981.287} C_VEL
LIN {X 0,Y 193.705,Z 222.888,A -85,B 0,C 180,E1 -21985.811,E2 -21985.811} C_VEL
LIN {X 0,Y 193.926,Z 223.771,A -85,B 0,C 180,E1 -21989.568,E2 -21989.568} C_VEL
LIN {X 0,Y 194.146,Z 225.087,A -85,B 0,C 180,E1 -21993.635,E2 -21993.635} C_VEL
LIN {X 0,Y 194.407,Z 226.85,A -85,B 0,C 180,E1 -21997.922,E2 -21997.922} C_VEL
LIN {X 0,Y 194.644,Z 228.198,A -85,B 0,C 180,E1 -22000.691,E2 -22000.691} C_VEL
LIN {X 0,Y 194.923,Z 229.923,A -85,B 0,C 180,E1 -22003.855,E2 -22003.855} C_VEL
LIN {X 0,Y 195.483,Z 233.185,A -85,B 0,C 180,E1 -22009.027,E2 -22009.027} C_VEL
LIN {X 0,Y 195.57,Z 233.627,A -85,B 0,C 180,E1 -22009.614,E2 -22009.614} C_VEL
LIN {X 0,Y 196.801,Z 236.835,A -85,B 0,C 180,E1 -22010.469,E2 -22010.469} C_VEL
LIN {X 0,Y 198.843,Z 239.822,A -85,B 0,C 180,E1 -22011.641,E2 -22011.641} C_VEL
LIN {X 0,Y 202.611,Z 248.289,A -85,B 0,C 180,E1 -22014.176,E2 -22014.176} C_VEL
LIN {X 0,Y 203.831,Z 253.194,A -85,B 0,C 180,E1 -22015.348,E2 -22015.348} C_VEL
LIN {X 0,Y 205.045,Z 263.67,A -85,B 0,C 180,E1 -22017.829,E2 -22017.829} C_VEL
LIN {X 0,Y 205.188,Z 271.899,A -85,B 0,C 180,E1 -22019.858,E2 -22019.858} C_VEL
LIN {X 0,Y 204.707,Z 279.272,A -85,B 0,C 180,E1 -22021.832,E2 -22021.832} C_VEL
LIN {X 0,Y 203.656,Z 285.912,A -85,B 0,C 180,E1 -22023.8,E2 -22023.8} C_VEL
LIN {X 0,Y 202.348,Z 290.748,A -85,B 0,C 180,E1 -22025.368,E2 -22025.368} C_VEL
LIN {X 0,Y 200.157,Z 296.031,A -85,B 0,C 180,E1 -22027.28,E2 -22027.28} C_VEL
LIN {X 0,Y 197.966,Z 300.517,A -85,B 0,C 180,E1 -22029.206,E2 -22029.206} C_VEL
LIN {X 0,Y 196.011,Z 304.277,A -85,B 0,C 180,E1 -22031.174,E2 -22031.174} C_VEL
LIN {X 0,Y 193.73,Z 308.592,A -85,B 0,C 180,E1 -22034.212,E2 -22034.212} C_VEL
LIN {X 0,Y 192.057,Z 311.672,A -85,B 0,C 180,E1 -22037.317,E2 -22037.317} C_VEL
LIN {X 0,Y 191.236,Z 313.089,A -85,B 0,C 180,E1 -22039.412,E2 -22039.412} C_VEL
LIN {X 0,Y 190.689,Z 314.045,A -85,B 0,C 180,E1 -22041.523,E2 -22041.523} C_VEL
LIN {X 0,Y 190.309,Z 314.426,A -85,B 0,C 180,E1 -22044.326,E2 -22044.326} C_VEL
LIN {X 0,Y 190.472,Z 313.763,A -85,B 0,C 180,E1 -22047.886,E2 -22047.886} C_VEL
LIN {X 0,Y 190.55,Z 312.689,A -85,B 0,C 180,E1 -22050,E2 -22050} C_VEL
LIN {X 0,Y 190.546,Z 311.082,A -85,B 0,C 180,E1 -22052.114,E2 -22052.114} C_VEL
LIN {X 0,Y 190.468,Z 309.739,A -85,B 0,C 180,E1 -22053.379,E2 -22053.379} C_VEL
LIN {X 0,Y 189.817,Z 307.76,A -85,B 0,C 180,E1 -22055.046,E2 -22055.046} C_VEL
LIN {X 0,Y 188.333,Z 305.408,A -85,B 0,C 180,E1 -22056.647,E2 -22056.647} C_VEL
LIN {X 0,Y 184.877,Z 299.22,A -85,B 0,C 180,E1 -22059.986,E2 -22059.986} C_VEL
LIN {X 0,Y 184.41,Z 295.163,A -85,B 0,C 180,E1 -22061.729,E2 -22061.729} C_VEL
LIN {X 0,Y 185.325,Z 288.268,A -85,B 0,C 180,E1 -22064.271,E2 -22064.271} C_VEL
LIN {X 0,Y 186.335,Z 280.988,A -85,B 0,C 180,E1 -22066.432,E2 -22066.432} C_VEL
LIN {X 0,Y 186.891,Z 276.806,A -85,B 0,C 180,E1 -22067.508,E2 -22067.508} C_VEL
LIN {X 0,Y 186.656,Z 267.999,A -85,B 0,C 180,E1 -22069.414,E2 -22069.414} C_VEL
LIN {X 0,Y 186.33,Z 258.958,A -85,B 0,C 180,E1 -22070.998,E2 -22070.998} C_VEL
LIN {X 0,Y 185.743,Z 249.164,A -85,B 0,C 180,E1 -22072.361,E2 -22072.361} C_VEL
LIN {X 0,Y 184.81,Z 237.251,A -85,B 0,C 180,E1 -22073.579,E2 -22073.579} C_VEL
LIN {X 0,Y 184.776,Z 236.321,A -85,B 0,C 180,E1 -22073.649,E2 -22073.649} C_VEL
LIN {X 0,Y 186.206,Z 230.46,A -85,B 0,C 180,E1 -22079.384,E2 -22079.384} C_VEL
LIN {X 0,Y 186.962,Z 228.035,A -85,B 0,C 180,E1 -22081.754,E2 -22081.754} C_VEL
LIN {X 0,Y 187.093,Z 225.533,A -85,B 0,C 180,E1 -22084.296,E2 -22084.296} C_VEL
LIN {X 0,Y 186.26,Z 221.406,A -85,B 0,C 180,E1 -22088.713,E2 -22088.713} C_VEL
LIN {X 0,Y 185.681,Z 218.17,A -85,B 0,C 180,E1 -22092.393,E2 -22092.393} C_VEL
LIN {X 0,Y 185.481,Z 218.189,A -85,B 0,C 180,E1 -22096.995,E2 -22096.995} C_VEL
LIN {X 0,Y 185.506,Z 218.188,A -85,B 0,C 180,E1 -22102.685,E2 -22102.685} C_VEL
LIN {X 0,Y 185.547,Z 218.185,A -85,B 0,C 180,E1 -22107.974,E2 -22107.974} C_VEL
LIN {X 0,Y 185.585,Z 218.178,A -85,B 0,C 180,E1 -22110.576,E2 -22110.576} C_VEL
LIN {X 0,Y 185.585,Z 218.178,A -85,B 0,C 180,E1 -22115.38,E2 -22115.38} C_VEL
LIN {X 0,Y 185.679,Z 218.165,A -85,B 0,C 180,E1 -22121.132,E2 -22121.132} C_VEL
LIN {X 0,Y 185.699,Z 218.164,A -85,B 0,C 180,E1 -22124.636,E2 -22124.636} C_VEL
LIN {X 0,Y 185.892,Z 218.139,A -85,B 0,C 180,E1 -22129.416,E2 -22129.416} C_VEL
LIN {X 0,Y 185.949,Z 218.136,A -85,B 0,C 180,E1 -22133.488,E2 -22133.488} C_VEL
LIN {X 0,Y 186.209,Z 218.097,A -85,B 0,C 180,E1 -22137.835,E2 -22137.835} C_VEL
LIN {X 0,Y 186.408,Z 218.075,A -85,B 0,C 180,E1 -22139.998,E2 -22139.998} C_VEL
LIN {X 0,Y 185.921,Z 218.137,A -85,B 0,C 180,E1 -22144.334,E2 -22144.334} C_VEL
LIN {X 0,Y 185.983,Z 218.129,A -85,B 0,C 180,E1 -22148.692,E2 -22148.692} C_VEL
LIN {X 0,Y 185.718,Z 218.161,A -85,B 0,C 180,E1 -22153.122,E2 -22153.122} C_VEL
LIN {X 0,Y 185.656,Z 218.169,A -85,B 0,C 180,E1 -22157.626,E2 -22157.626} C_VEL
LIN {X 0,Y 185.574,Z 218.18,A -85,B 0,C 180,E1 -22162.252,E2 -22162.252} C_VEL
LIN {X 0,Y 185.56,Z 218.183,A -85,B 0,C 180,E1 -22167.03,E2 -22167.03} C_VEL
LIN {X 0,Y 185.578,Z 218.179,A -85,B 0,C 180,E1 -22169.491,E2 -22169.491} C_VEL
LIN {X 0,Y 185.517,Z 218.188,A -85,B 0,C 180,E1 -22174.625,E2 -22174.625} C_VEL
LIN {X 0,Y 185.542,Z 218.184,A -85,B 0,C 180,E1 -22177.302,E2 -22177.302} C_VEL
LIN {X 0,Y 185.482,Z 218.189,A -85,B 0,C 180,E1 -22180.728,E2 -22180.728} C_VEL
LIN {X 0,Y 185.457,Z 218.195,A -85,B 0,C 180,E1 -22186.053,E2 -22186.053} C_VEL
LIN {X 0,Y 185.464,Z 218.194,A -85,B 0,C 180,E1 -22189.894,E2 -22189.894} C_VEL
LIN {X 0,Y 185.502,Z 218.189,A -85,B 0,C 180,E1 -22192.71,E2 -22192.71} C_VEL
LIN {X 0,Y 185.542,Z 218.184,A -85,B 0,C 180,E1 -22197.974,E2 -22197.974} C_VEL
LIN {X 0,Y 185.577,Z 218.18,A -85,B 0,C 180,E1 -22200.574,E2 -22200.574} C_VEL
LIN {X 0,Y 185.582,Z 218.177,A -85,B 0,C 180,E1 -22205.381,E2 -22205.381} C_VEL
LIN {X 0,Y 185.669,Z 218.17,A -85,B 0,C 180,E1 -22211.132,E2 -22211.132} C_VEL
LIN {X 0,Y 185.758,Z 218.159,A -85,B 0,C 180,E1 -22216.879,E2 -22216.879} C_VEL
LIN {X 0,Y 186.003,Z 218.124,A -85,B 0,C 180,E1 -22221.307,E2 -22221.307} C_VEL
LIN {X 0,Y 186.201,Z 218.101,A -85,B 0,C 180,E1 -22227.836,E2 -22227.836} C_VEL
LIN {X 0,Y 186.4,Z 218.074,A -85,B 0,C 180,E1 -22230,E2 -22230} C_VEL
LIN {X 0,Y 185.918,Z 218.139,A -85,B 0,C 180,E1 -22234.335,E2 -22234.335} C_VEL
LIN {X 0,Y 185.963,Z 218.13,A -85,B 0,C 180,E1 -22238.694,E2 -22238.694} C_VEL
LIN {X 0,Y 185.429,Z 218.198,A -85,B 0,C 180,E1 -22243.144,E2 -22243.144} C_VEL
LIN {X 0,Y 185.008,Z 218.312,A -85,B 0,C 180,E1 -22246.269,E2 -22246.269} C_VEL
LIN {X 0,Y 184.257,Z 223.122,A -85,B 0,C 180,E1 -22252.348,E2 -22252.348} C_VEL
LIN {X 0,Y 186.024,Z 233.914,A -85,B 0,C 180,E1 -22253.559,E2 -22253.559} C_VEL
LIN {X 0,Y 187.337,Z 243.52,A -85,B 0,C 180,E1 -22254.964,E2 -22254.964} C_VEL
LIN {X 0,Y 188.369,Z 252.5,A -85,B 0,C 180,E1 -22256.597,E2 -22256.597} C_VEL
LIN {X 0,Y 188.154,Z 257.009,A -85,B 0,C 180,E1 -22257.531,E2 -22257.531} C_VEL
LIN {X 0,Y 187.104,Z 264.204,A -85,B 0,C 180,E1 -22259.229,E2 -22259.229} C_VEL
LIN {X 0,Y 185.952,Z 271.856,A -85,B 0,C 180,E1 -22261.455,E2 -22261.455} C_VEL
LIN {X 0,Y 184.917,Z 278.91,A -85,B 0,C 180,E1 -22264.016,E2 -22264.016} C_VEL
LIN {X 0,Y 184.044,Z 284.647,A -85,B 0,C 180,E1 -22266.691,E2 -22266.691} C_VEL
LIN {X 0,Y 183.533,Z 288.388,A -85,B 0,C 180,E1 -22268.83,E2 -22268.83} C_VEL
LIN {X 0,Y 183.056,Z 292.506,A -85,B 0,C 180,E1 -22271.918,E2 -22271.918} C_VEL
LIN {X 0,Y 182.96,Z 294.448,A -85,B 0,C 180,E1 -22273.743,E2 -22273.743} C_VEL
LIN {X 0,Y 183.072,Z 296.703,A -85,B 0,C 180,E1 -22276.835,E2 -22276.835} C_VEL
LIN {X 0,Y 183.57,Z 297.923,A -85,B 0,C 180,E1 -22279.969,E2 -22279.969} C_VEL
LIN {X 0,Y 184.547,Z 298.101,A -85,B 0,C 180,E1 -22283.104,E2 -22283.104} C_VEL
LIN {X 0,Y 186.001,Z 297.223,A -85,B 0,C 180,E1 -22286.228,E2 -22286.228} C_VEL
LIN {X 0,Y 187.897,Z 295.248,A -85,B 0,C 180,E1 -22289.347,E2 -22289.347} C_VEL
LIN {X 0,Y 190.288,Z 291.972,A -85,B 0,C 180,E1 -22292.424,E2 -22292.424} C_VEL
LIN {X 0,Y 193.221,Z 287.32,A -85,B 0,C 180,E1 -22295.411,E2 -22295.411} C_VEL
LIN {X 0,Y 195.665,Z 282.92,A -85,B 0,C 180,E1 -22297.566,E2 -22297.566} C_VEL
LIN {X 0,Y 198.65,Z 277.035,A -85,B 0,C 180,E1 -22299.824,E2 -22299.824} C_VEL
LIN {X 0,Y 200.121,Z 273.333,A -85,B 0,C 180,E1 -22301.047,E2 -22301.047} C_VEL
LIN {X 0,Y 200.553,Z 267.526,A -85,B 0,C 180,E1 -22303.144,E2 -22303.144} C_VEL
LIN {X 0,Y 200.316,Z 260.812,A -85,B 0,C 180,E1 -22305.411,E2 -22305.411} C_VEL
LIN {X 0,Y 199.273,Z 253.482,A -85,B 0,C 180,E1 -22307.785,E2 -22307.785} C_VEL
LIN {X 0,Y 197.793,Z 247.56,A -85,B 0,C 180,E1 -22309.768,E2 -22309.768} C_VEL
LIN {X 0,Y 195.453,Z 240.898,A -85,B 0,C 180,E1 -22312.082,E2 -22312.082} C_VEL
LIN {X 0,Y 193.443,Z 236.611,A -85,B 0,C 180,E1 -22313.745,E2 -22313.745} C_VEL
LIN {X 0,Y 191.278,Z 233.079,A -85,B 0,C 180,E1 -22315.326,E2 -22315.326} C_VEL
LIN {X 0,Y 190.392,Z 231.434,A -85,B 0,C 180,E1 -22316.007,E2 -22316.007} C_VEL
LIN {X 0,Y 188.335,Z 228.461,A -85,B 0,C 180,E1 -22317.529,E2 -22317.529} C_VEL
LIN {X 0,Y 187.752,Z 226.572,A -85,B 0,C 180,E1 -22318.192,E2 -22318.192} C_VEL
LIN {X 0,Y 187.821,Z 225.998,A -85,B 0,C 180,E1 -22320.002,E2 -22320.002} C_VEL
LIN {X 0,Y 187.306,Z 225.027,A -85,B 0,C 180,E1 -22324.305,E2 -22324.305} C_VEL
LIN {X 0,Y 187.178,Z 224.27,A -85,B 0,C 180,E1 -22328.64,E2 -22328.64} C_VEL
LIN {X 0,Y 186.878,Z 223.902,A -85,B 0,C 180,E1 -22333.042,E2 -22333.042} C_VEL
LIN {X 0,Y 186.803,Z 223.86,A -85,B 0,C 180,E1 -22337.518,E2 -22337.518} C_VEL
LIN {X 0,Y 186.762,Z 224.231,A -85,B 0,C 180,E1 -22342.107,E2 -22342.107} C_VEL
LIN {X 0,Y 186.92,Z 225.013,A -85,B 0,C 180,E1 -22346.822,E2 -22346.822} C_VEL
LIN {X 0,Y 187.097,Z 225.85,A -85,B 0,C 180,E1 -22350.237,E2 -22350.237} C_VEL
LIN {X 0,Y 187.332,Z 227.207,A -85,B 0,C 180,E1 -22354.376,E2 -22354.376} C_VEL
LIN {X 0,Y 187.638,Z 229.403,A -85,B 0,C 180,E1 -22359.551,E2 -22359.551} C_VEL
LIN {X 0,Y 188.07,Z 232.144,A -85,B 0,C 180,E1 -22364.764,E2 -22364.764} C_VEL
LIN {X 0,Y 188.28,Z 233.229,A -85,B 0,C 180,E1 -22366.323,E2 -22366.323} C_VEL
LIN {X 0,Y 189.616,Z 236.45,A -85,B 0,C 180,E1 -22367.411,E2 -22367.411} C_VEL
LIN {X 0,Y 191.765,Z 239.431,A -85,B 0,C 180,E1 -22368.851,E2 -22368.851} C_VEL
LIN {X 0,Y 193.045,Z 242.526,A -85,B 0,C 180,E1 -22369.867,E2 -22369.867} C_VEL
LIN {X 0,Y 194.659,Z 245.156,A -85,B 0,C 180,E1 -22370.92,E2 -22370.92} C_VEL
LIN {X 0,Y 197.503,Z 252.085,A -85,B 0,C 180,E1 -22373.192,E2 -22373.192} C_VEL
LIN {X 0,Y 198.559,Z 257.429,A -85,B 0,C 180,E1 -22374.657,E2 -22374.657} C_VEL
LIN {X 0,Y 199.246,Z 265.436,A -85,B 0,C 180,E1 -22376.7,E2 -22376.7} C_VEL
LIN {X 0,Y 199.121,Z 274.742,A -85,B 0,C 180,E1 -22379.188,E2 -22379.188} C_VEL
LIN {X 0,Y 197.939,Z 283.97,A -85,B 0,C 180,E1 -22381.937,E2 -22381.937} C_VEL
LIN {X 0,Y 196.43,Z 290.145,A -85,B 0,C 180,E1 -22384.01,E2 -22384.01} C_VEL
LIN {X 0,Y 194.313,Z 295.437,A -85,B 0,C 180,E1 -22385.99,E2 -22385.99} C_VEL
LIN {X 0,Y 191.375,Z 300.9,A -85,B 0,C 180,E1 -22388.455,E2 -22388.455} C_VEL
LIN {X 0,Y 188.464,Z 306.025,A -85,B 0,C 180,E1 -22391.52,E2 -22391.52} C_VEL
LIN {X 0,Y 186.259,Z 309.846,A -85,B 0,C 180,E1 -22394.685,E2 -22394.685} C_VEL
LIN {X 0,Y 185.112,Z 311.627,A -85,B 0,C 180,E1 -22396.833,E2 -22396.833} C_VEL
LIN {X 0,Y 184.239,Z 312.926,A -85,B 0,C 180,E1 -22399.005,E2 -22399.005} C_VEL
LIN {X 0,Y 183.661,Z 313.767,A -85,B 0,C 180,E1 -22401.196,E2 -22401.196} C_VEL
LIN {X 0,Y 183.307,Z 314.145,A -85,B 0,C 180,E1 -22403.396,E2 -22403.396} C_VEL
LIN {X 0,Y 183.207,Z 313.922,A -85,B 0,C 180,E1 -22405.875,E2 -22405.875} C_VEL
LIN {X 0,Y 183.402,Z 313.266,A -85,B 0,C 180,E1 -22407.804,E2 -22407.804} C_VEL
LIN {X 0,Y 183.487,Z 312.089,A -85,B 0,C 180,E1 -22410,E2 -22410} C_VEL
LIN {X 0,Y 183.481,Z 310.376,A -85,B 0,C 180,E1 -22412.196,E2 -22412.196} C_VEL
LIN {X 0,Y 183.431,Z 307.251,A -85,B 0,C 180,E1 -22415.003,E2 -22415.003} C_VEL
LIN {X 0,Y 183.614,Z 303.249,A -85,B 0,C 180,E1 -22417.699,E2 -22417.699} C_VEL
LIN {X 0,Y 184.093,Z 298.012,A -85,B 0,C 180,E1 -22420.448,E2 -22420.448} C_VEL
LIN {X 0,Y 184.41,Z 295.163,A -85,B 0,C 180,E1 -22421.729,E2 -22421.729} C_VEL
LIN {X 0,Y 184.265,Z 291.562,A -85,B 0,C 180,E1 -22423.142,E2 -22423.142} C_VEL
LIN {X 0,Y 183.358,Z 287.708,A -85,B 0,C 180,E1 -22424.504,E2 -22424.504} C_VEL
LIN {X 0,Y 180.8,Z 279.223,A -85,B 0,C 180,E1 -22427.062,E2 -22427.062} C_VEL
LIN {X 0,Y 179.79,Z 272.944,A -85,B 0,C 180,E1 -22428.647,E2 -22428.647} C_VEL
LIN {X 0,Y 179.5,Z 263.402,A -85,B 0,C 180,E1 -22430.633,E2 -22430.633} C_VEL
LIN {X 0,Y 178.898,Z 252.468,A -85,B 0,C 180,E1 -22432.37,E2 -22432.37} C_VEL
LIN {X 0,Y 178.276,Z 242.36,A -85,B 0,C 180,E1 -22433.576,E2 -22433.576} C_VEL
LIN {X 0,Y 177.752,Z 236.071,A -85,B 0,C 180,E1 -22434.192,E2 -22434.192} C_VEL
LIN {X 0,Y 179.082,Z 231.054,A -85,B 0,C 180,E1 -22439.309,E2 -22439.309} C_VEL
LIN {X 0,Y 180.085,Z 227.341,A -85,B 0,C 180,E1 -22443.118,E2 -22443.118} C_VEL
LIN {X 0,Y 179.78,Z 224.757,A -85,B 0,C 180,E1 -22445.901,E2 -22445.901} C_VEL
LIN {X 0,Y 178.687,Z 219.303,A -85,B 0,C 180,E1 -22452.151,E2 -22452.151} C_VEL
LIN {X 0,Y 178.547,Z 219.055,A -85,B 0,C 180,E1 -22453.4,E2 -22453.4} C_VEL
LIN {X 0,Y 178.409,Z 219.074,A -85,B 0,C 180,E1 -22458.458,E2 -22458.458} C_VEL
LIN {X 0,Y 178.425,Z 219.07,A -85,B 0,C 180,E1 -22463.782,E2 -22463.782} C_VEL
LIN {X 0,Y 178.49,Z 219.062,A -85,B 0,C 180,E1 -22466.546,E2 -22466.546} C_VEL
LIN {X 0,Y 178.526,Z 219.06,A -85,B 0,C 180,E1 -22470.006,E2 -22470.006} C_VEL
LIN {X 0,Y 178.524,Z 219.057,A -85,B 0,C 180,E1 -22474.885,E2 -22474.885} C_VEL
LIN {X 0,Y 178.627,Z 219.043,A -85,B 0,C 180,E1 -22480.783,E2 -22480.783} C_VEL
LIN {X 0,Y 178.662,Z 219.041,A -85,B 0,C 180,E1 -22486.346,E2 -22486.346} C_VEL
LIN {X 0,Y 178.914,Z 219.007,A -85,B 0,C 180,E1 -22490.958,E2 -22490.958} C_VEL
LIN {X 0,Y 179.155,Z 218.976,A -85,B 0,C 180,E1 -22497.75,E2 -22497.75} C_VEL
LIN {X 0,Y 179.371,Z 218.952,A -85,B 0,C 180,E1 -22499.998,E2 -22499.998} C_VEL
LIN {X 0,Y 178.868,Z 219.015,A -85,B 0,C 180,E1 -22504.505,E2 -22504.505} C_VEL
LIN {X 0,Y 178.912,Z 219.012,A -85,B 0,C 180,E1 -22509.038,E2 -22509.038} C_VEL
LIN {X 0,Y 178.644,Z 219.041,A -85,B 0,C 180,E1 -22513.651,E2 -22513.651} C_VEL
LIN {X 0,Y 178.59,Z 219.051,A -85,B 0,C 180,E1 -22519.183,E2 -22519.183} C_VEL
LIN {X 0,Y 178.519,Z 219.058,A -85,B 0,C 180,E1 -22525.112,E2 -22525.112} C_VEL
LIN {X 0,Y 178.522,Z 219.059,A -85,B 0,C 180,E1 -22529.992,E2 -22529.992} C_VEL
LIN {X 0,Y 178.494,Z 219.063,A -85,B 0,C 180,E1 -22534.223,E2 -22534.223} C_VEL
LIN {X 0,Y 178.416,Z 219.069,A -85,B 0,C 180,E1 -22539.066,E2 -22539.066} C_VEL
LIN {X 0,Y 178.4,Z 219.074,A -85,B 0,C 180,E1 -22542.041,E2 -22542.041} C_VEL
LIN {X 0,Y 178.395,Z 219.075,A -85,B 0,C 180,E1 -22545.16,E2 -22545.16} C_VEL
LIN {X 0,Y 178.399,Z 219.07,A -85,B 0,C 180,E1 -22548.457,E2 -22548.457} C_VEL
LIN {X 0,Y 178.418,Z 219.073,A -85,B 0,C 180,E1 -22553.781,E2 -22553.781} C_VEL
LIN {X 0,Y 178.483,Z 219.059,A -85,B 0,C 180,E1 -22556.545,E2 -22556.545} C_VEL
LIN {X 0,Y 178.518,Z 219.06,A -85,B 0,C 180,E1 -22560.005,E2 -22560.005} C_VEL
LIN {X 0,Y 178.529,Z 219.055,A -85,B 0,C 180,E1 -22564.874,E2 -22564.874} C_VEL
LIN {X 0,Y 178.617,Z 219.047,A -85,B 0,C 180,E1 -22570.783,E2 -22570.783} C_VEL
LIN {X 0,Y 178.675,Z 219.039,A -85,B 0,C 180,E1 -22576.349,E2 -22576.349} C_VEL
LIN {X 0,Y 178.953,Z 219.003,A -85,B 0,C 180,E1 -22580.961,E2 -22580.961} C_VEL
LIN {X 0,Y 179.147,Z 218.98,A -85,B 0,C 180,E1 -22587.751,E2 -22587.751} C_VEL
LIN {X 0,Y 179.363,Z 218.95,A -85,B 0,C 180,E1 -22590,E2 -22590} C_VEL
LIN {X 0,Y 178.866,Z 219.018,A -85,B 0,C 180,E1 -22594.507,E2 -22594.507} C_VEL
LIN {X 0,Y 178.879,Z 219.012,A -85,B 0,C 180,E1 -22599.042,E2 -22599.042} C_VEL
LIN {X 0,Y 178.294,Z 219.087,A -85,B 0,C 180,E1 -22603.68,E2 -22603.68} C_VEL
LIN {X 0,Y 177.902,Z 219.17,A -85,B 0,C 180,E1 -22606.342,E2 -22606.342} C_VEL
LIN {X 0,Y 177.241,Z 223.42,A -85,B 0,C 180,E1 -22611.823,E2 -22611.823} C_VEL
LIN {X 0,Y 179.005,Z 234.419,A -85,B 0,C 180,E1 -22613.117,E2 -22613.117} C_VEL
LIN {X 0,Y 180.208,Z 243.387,A -85,B 0,C 180,E1 -22614.479,E2 -22614.479} C_VEL
LIN {X 0,Y 181.238,Z 252.205,A -85,B 0,C 180,E1 -22616.132,E2 -22616.132} C_VEL
LIN {X 0,Y 181.318,Z 256.063,A -85,B 0,C 180,E1 -22616.943,E2 -22616.943} C_VEL
LIN {X 0,Y 180.12,Z 264.071,A -85,B 0,C 180,E1 -22618.872,E2 -22618.872} C_VEL
LIN {X 0,Y 179.008,Z 271.29,A -85,B 0,C 180,E1 -22621.017,E2 -22621.017} C_VEL
LIN {X 0,Y 177.961,Z 278.223,A -85,B 0,C 180,E1 -22623.565,E2 -22623.565} C_VEL
LIN {X 0,Y 176.969,Z 284.647,A -85,B 0,C 180,E1 -22626.562,E2 -22626.562} C_VEL
LIN {X 0,Y 176.27,Z 289.626,A -85,B 0,C 180,E1 -22629.637,E2 -22629.637} C_VEL
LIN {X 0,Y 175.894,Z 293.463,A -85,B 0,C 180,E1 -22632.785,E2 -22632.785} C_VEL
LIN {X 0,Y 175.916,Z 296.218,A -85,B 0,C 180,E1 -22635.981,E2 -22635.981} C_VEL
LIN {X 0,Y 176.315,Z 297.938,A -85,B 0,C 180,E1 -22639.23,E2 -22639.23} C_VEL
LIN {X 0,Y 177.204,Z 298.575,A -85,B 0,C 180,E1 -22642.486,E2 -22642.486} C_VEL
LIN {X 0,Y 179.06,Z 297.745,A -85,B 0,C 180,E1 -22646.671,E2 -22646.671} C_VEL
LIN {X 0,Y 180.892,Z 296.066,A -85,B 0,C 180,E1 -22649.666,E2 -22649.666} C_VEL
LIN {X 0,Y 183.154,Z 293.405,A -85,B 0,C 180,E1 -22652.585,E2 -22652.585} C_VEL
LIN {X 0,Y 185.899,Z 289.644,A -85,B 0,C 180,E1 -22655.429,E2 -22655.429} C_VEL
LIN {X 0,Y 189.119,Z 284.381,A -85,B 0,C 180,E1 -22658.285,E2 -22658.285} C_VEL
LIN {X 0,Y 191.653,Z 279.89,A -85,B 0,C 180,E1 -22660.198,E2 -22660.198} C_VEL
LIN {X 0,Y 193.729,Z 275.723,A -85,B 0,C 180,E1 -22661.708,E2 -22661.708} C_VEL
LIN {X 0,Y 194.432,Z 270.508,A -85,B 0,C 180,E1 -22663.734,E2 -22663.734} C_VEL
LIN {X 0,Y 194.428,Z 263.193,A -85,B 0,C 180,E1 -22666.413,E2 -22666.413} C_VEL
LIN {X 0,Y 193.589,Z 255.905,A -85,B 0,C 180,E1 -22669.014,E2 -22669.014} C_VEL
LIN {X 0,Y 191.768,Z 248.621,A -85,B 0,C 180,E1 -22671.691,E2 -22671.691} C_VEL
LIN {X 0,Y 188.914,Z 241.479,A -85,B 0,C 180,E1 -22674.665,E2 -22674.665} C_VEL
LIN {X 0,Y 186.58,Z 237.027,A -85,B 0,C 180,E1 -22676.763,E2 -22676.763} C_VEL
LIN {X 0,Y 184.665,Z 233.618,A -85,B 0,C 180,E1 -22678.503,E2 -22678.503} C_VEL
LIN {X 0,Y 184.132,Z 232.394,A -85,B 0,C 180,E1 -22679.045,E2 -22679.045} C_VEL
LIN {X 0,Y 181.412,Z 229.012,A -85,B 0,C 180,E1 -22681.388,E2 -22681.388} C_VEL
LIN {X 0,Y 180.71,Z 227.22,A -85,B 0,C 180,E1 -22682.231,E2 -22682.231} C_VEL
LIN {X 0,Y 180.295,Z 226.098,A -85,B 0,C 180,E1 -22688.972,E2 -22688.972} C_VEL
LIN {X 0,Y 180.021,Z 225.793,A -85,B 0,C 180,E1 -22693.549,E2 -22693.549} C_VEL
LIN {X 0,Y 179.957,Z 225.824,A -85,B 0,C 180,E1 -22698.208,E2 -22698.208} C_VEL
LIN {X 0,Y 179.945,Z 226.282,A -85,B 0,C 180,E1 -22702.991,E2 -22702.991} C_VEL
LIN {X 0,Y 180.067,Z 226.781,A -85,B 0,C 180,E1 -22706.145,E2 -22706.145} C_VEL
LIN {X 0,Y 180.257,Z 227.946,A -85,B 0,C 180,E1 -22710.935,E2 -22710.935} C_VEL
LIN {X 0,Y 180.523,Z 229.561,A -85,B 0,C 180,E1 -22715.732,E2 -22715.732} C_VEL
LIN {X 0,Y 180.712,Z 230.912,A -85,B 0,C 180,E1 -22718.94,E2 -22718.94} C_VEL
LIN {X 0,Y 181.007,Z 232.57,A -85,B 0,C 180,E1 -22722.162,E2 -22722.162} C_VEL
LIN {X 0,Y 182.153,Z 235.539,A -85,B 0,C 180,E1 -22723.375,E2 -22723.375} C_VEL
LIN {X 0,Y 184.815,Z 239.255,A -85,B 0,C 180,E1 -22725.595,E2 -22725.595} C_VEL
LIN {X 0,Y 186.117,Z 242.29,A -85,B 0,C 180,E1 -22726.773,E2 -22726.773} C_VEL
LIN {X 0,Y 187.594,Z 244.412,A -85,B 0,C 180,E1 -22727.871,E2 -22727.871} C_VEL
LIN {X 0,Y 189.247,Z 248.393,A -85,B 0,C 180,E1 -22729.437,E2 -22729.437} C_VEL
LIN {X 0,Y 191.566,Z 253.483,A -85,B 0,C 180,E1 -22731.415,E2 -22731.415} C_VEL
LIN {X 0,Y 192.828,Z 257.846,A -85,B 0,C 180,E1 -22732.876,E2 -22732.876} C_VEL
LIN {X 0,Y 193.414,Z 264.78,A -85,B 0,C 180,E1 -22734.834,E2 -22734.834} C_VEL
LIN {X 0,Y 193.329,Z 273.539,A -85,B 0,C 180,E1 -22737.319,E2 -22737.319} C_VEL
LIN {X 0,Y 192.38,Z 281.813,A -85,B 0,C 180,E1 -22739.847,E2 -22739.847} C_VEL
LIN {X 0,Y 190.516,Z 289.663,A -85,B 0,C 180,E1 -22742.596,E2 -22742.596} C_VEL
LIN {X 0,Y 188.482,Z 294.856,A -85,B 0,C 180,E1 -22744.609,E2 -22744.609} C_VEL
LIN {X 0,Y 185.942,Z 299.406,A -85,B 0,C 180,E1 -22746.618,E2 -22746.618} C_VEL
LIN {X 0,Y 182.658,Z 304.762,A -85,B 0,C 180,E1 -22749.74,E2 -22749.74} C_VEL
LIN {X 0,Y 180.077,Z 308.78,A -85,B 0,C 180,E1 -22752.98,E2 -22752.98} C_VEL
LIN {X 0,Y 178.183,Z 311.593,A -85,B 0,C 180,E1 -22756.311,E2 -22756.311} C_VEL
LIN {X 0,Y 177.262,Z 312.766,A -85,B 0,C 180,E1 -22758.566,E2 -22758.566} C_VEL
LIN {X 0,Y 176.631,Z 313.489,A -85,B 0,C 180,E1 -22760.842,E2 -22760.842} C_VEL
LIN {X 0,Y 176.245,Z 313.763,A -85,B 0,C 180,E1 -22763.13,E2 -22763.13} C_VEL
LIN {X 0,Y 176.144,Z 313.397,A -85,B 0,C 180,E1 -22765.948,E2 -22765.948} C_VEL
LIN {X 0,Y 176.332,Z 312.758,A -85,B 0,C 180,E1 -22767.716,E2 -22767.716} C_VEL
LIN {X 0,Y 176.426,Z 311.461,A -85,B 0,C 180,E1 -22770,E2 -22770} C_VEL
LIN {X 0,Y 176.418,Z 309.626,A -85,B 0,C 180,E1 -22772.284,E2 -22772.284} C_VEL
LIN {X 0,Y 176.361,Z 306.712,A -85,B 0,C 180,E1 -22774.945,E2 -22774.945} C_VEL
LIN {X 0,Y 176.594,Z 302.245,A -85,B 0,C 180,E1 -22778.007,E2 -22778.007} C_VEL
LIN {X 0,Y 177.1,Z 296.864,A -85,B 0,C 180,E1 -22780.866,E2 -22780.866} C_VEL
LIN {X 0,Y 177.982,Z 290.102,A -85,B 0,C 180,E1 -22783.705,E2 -22783.705} C_VEL
LIN {X 0,Y 179.211,Z 281.295,A -85,B 0,C 180,E1 -22786.519,E2 -22786.519} C_VEL
LIN {X 0,Y 179.834,Z 277.234,A -85,B 0,C 180,E1 -22787.631,E2 -22787.631} C_VEL
LIN {X 0,Y 179.79,Z 272.944,A -85,B 0,C 180,E1 -22788.647,E2 -22788.647} C_VEL
LIN {X 0,Y 178.914,Z 268.209,A -85,B 0,C 180,E1 -22789.738,E2 -22789.738} C_VEL
LIN {X 0,Y 175.791,Z 260.286,A -85,B 0,C 180,E1 -22791.391,E2 -22791.391} C_VEL
LIN {X 0,Y 172.577,Z 251.975,A -85,B 0,C 180,E1 -22792.85,E2 -22792.85} C_VEL
LIN {X 0,Y 171.565,Z 246.587,A -85,B 0,C 180,E1 -22793.608,E2 -22793.608} C_VEL
LIN {X 0,Y 170.779,Z 235.81,A -85,B 0,C 180,E1 -22794.747,E2 -22794.747} C_VEL
LIN {X 0,Y 171.994,Z 231.479,A -85,B 0,C 180,E1 -22799.364,E2 -22799.364} C_VEL
LIN {X 0,Y 173.011,Z 227.842,A -85,B 0,C 180,E1 -22803.257,E2 -22803.257} C_VEL
LIN {X 0,Y 172.771,Z 225.817,A -85,B 0,C 180,E1 -22805.552,E2 -22805.552} C_VEL
LIN {X 0,Y 171.85,Z 221.32,A -85,B 0,C 180,E1 -22810.87,E2 -22810.87} C_VEL
LIN {X 0,Y 171.577,Z 219.925,A -85,B 0,C 180,E1 -22812.77,E2 -22812.77} C_VEL
LIN {X 0,Y 171.34,Z 219.953,A -85,B 0,C 180,E1 -22818.981,E2 -22818.981} C_VEL
LIN {X 0,Y 171.388,Z 219.95,A -85,B 0,C 180,E1 -22822.039,E2 -22822.039} C_VEL
LIN {X 0,Y 171.402,Z 219.941,A -85,B 0,C 180,E1 -22825.092,E2 -22825.092} C_VEL
LIN {X 0,Y 171.452,Z 219.939,A -85,B 0,C 180,E1 -22830.533,E2 -22830.533} C_VEL
LIN {X 0,Y 171.45,Z 219.941,A -85,B 0,C 180,E1 -22835.799,E2 -22835.799} C_VEL
LIN {X 0,Y 171.583,Z 219.92,A -85,B 0,C 180,E1 -22840.87,E2 -22840.87} C_VEL
LIN {X 0,Y 171.58,Z 219.925,A -85,B 0,C 180,E1 -22845.771,E2 -22845.771} C_VEL
LIN {X 0,Y 171.851,Z 219.886,A -85,B 0,C 180,E1 -22850.583,E2 -22850.583} C_VEL
LIN {X 0,Y 171.817,Z 219.896,A -85,B 0,C 180,E1 -22855.306,E2 -22855.306} C_VEL
LIN {X 0,Y 172.334,Z 219.828,A -85,B 0,C 180,E1 -22859.998,E2 -22859.998} C_VEL
LIN {X 0,Y 171.816,Z 219.895,A -85,B 0,C 180,E1 -22864.69,E2 -22864.69} C_VEL
LIN {X 0,Y 171.849,Z 219.891,A -85,B 0,C 180,E1 -22869.413,E2 -22869.413} C_VEL
LIN {X 0,Y 171.559,Z 219.924,A -85,B 0,C 180,E1 -22874.226,E2 -22874.226} C_VEL
LIN {X 0,Y 171.515,Z 219.932,A -85,B 0,C 180,E1 -22879.532,E2 -22879.532} C_VEL
LIN {X 0,Y 171.458,Z 219.937,A -85,B 0,C 180,E1 -22885.607,E2 -22885.607} C_VEL
LIN {X 0,Y 171.441,Z 219.938,A -85,B 0,C 180,E1 -22890.585,E2 -22890.585} C_VEL
LIN {X 0,Y 171.405,Z 219.945,A -85,B 0,C 180,E1 -22895.029,E2 -22895.029} C_VEL
LIN {X 0,Y 171.378,Z 219.946,A -85,B 0,C 180,E1 -22898.815,E2 -22898.815} C_VEL
LIN {X 0,Y 171.324,Z 219.957,A -85,B 0,C 180,E1 -22904.213,E2 -22904.213} C_VEL
LIN {X 0,Y 171.331,Z 219.95,A -85,B 0,C 180,E1 -22908.98,E2 -22908.98} C_VEL
LIN {X 0,Y 171.383,Z 219.95,A -85,B 0,C 180,E1 -22912.039,E2 -22912.039} C_VEL
LIN {X 0,Y 171.394,Z 219.946,A -85,B 0,C 180,E1 -22915.09,E2 -22915.09} C_VEL
LIN {X 0,Y 171.444,Z 219.94,A -85,B 0,C 180,E1 -22920.533,E2 -22920.533} C_VEL
LIN {X 0,Y 171.452,Z 219.938,A -85,B 0,C 180,E1 -22925.8,E2 -22925.8} C_VEL
LIN {X 0,Y 171.573,Z 219.925,A -85,B 0,C 180,E1 -22930.87,E2 -22930.87} C_VEL
LIN {X 0,Y 171.588,Z 219.922,A -85,B 0,C 180,E1 -22935.773,E2 -22935.773} C_VEL
LIN {X 0,Y 171.882,Z 219.885,A -85,B 0,C 180,E1 -22940.586,E2 -22940.586} C_VEL
LIN {X 0,Y 171.815,Z 219.895,A -85,B 0,C 180,E1 -22945.307,E2 -22945.307} C_VEL
LIN {X 0,Y 172.326,Z 219.827,A -85,B 0,C 180,E1 -22950,E2 -22950} C_VEL
LIN {X 0,Y 171.814,Z 219.897,A -85,B 0,C 180,E1 -22954.692,E2 -22954.692} C_VEL
LIN {X 0,Y 171.864,Z 219.886,A -85,B 0,C 180,E1 -22957.046,E2 -22957.046} C_VEL
LIN {X 0,Y 171.665,Z 219.914,A -85,B 0,C 180,E1 -22960.729,E2 -22960.729} C_VEL
LIN {X 0,Y 170.856,Z 220.014,A -85,B 0,C 180,E1 -22966.273,E2 -22966.273} C_VEL
LIN {X 0,Y 170.183,Z 223.452,A -85,B 0,C 180,E1 -22971.182,E2 -22971.182} C_VEL
LIN {X 0,Y 171.902,Z 234.229,A -85,B 0,C 180,E1 -22972.537,E2 -22972.537} C_VEL
LIN {X 0,Y 173.11,Z 243.235,A -85,B 0,C 180,E1 -22973.952,E2 -22973.952} C_VEL
LIN {X 0,Y 174.005,Z 250.874,A -85,B 0,C 180,E1 -22975.413,E2 -22975.413} C_VEL
LIN {X 0,Y 174.406,Z 255.111,A -85,B 0,C 180,E1 -22976.312,E2 -22976.312} C_VEL
LIN {X 0,Y 173.332,Z 262.756,A -85,B 0,C 180,E1 -22978.151,E2 -22978.151} C_VEL
LIN {X 0,Y 172.084,Z 270.616,A -85,B 0,C 180,E1 -22980.506,E2 -22980.506} C_VEL
LIN {X 0,Y 171.025,Z 277.309,A -85,B 0,C 180,E1 -22982.989,E2 -22982.989} C_VEL
LIN {X 0,Y 170.011,Z 283.782,A -85,B 0,C 180,E1 -22985.983,E2 -22985.983} C_VEL
LIN {X 0,Y 169.256,Z 289.167,A -85,B 0,C 180,E1 -22989.231,E2 -22989.231} C_VEL
LIN {X 0,Y 168.877,Z 292.405,A -85,B 0,C 180,E1 -22991.748,E2 -22991.748} C_VEL
LIN {X 0,Y 168.775,Z 295.545,A -85,B 0,C 180,E1 -22995.064,E2 -22995.064} C_VEL
LIN {X 0,Y 169.074,Z 297.645,A -85,B 0,C 180,E1 -22998.436,E2 -22998.436} C_VEL
LIN {X 0,Y 169.853,Z 298.721,A -85,B 0,C 180,E1 -23001.828,E2 -23001.828} C_VEL
LIN {X 0,Y 171.178,Z 298.76,A -85,B 0,C 180,E1 -23005.198,E2 -23005.198} C_VEL
LIN {X 0,Y 172.963,Z 297.743,A -85,B 0,C 180,E1 -23008.571,E2 -23008.571} C_VEL
LIN {X 0,Y 175.319,Z 295.557,A -85,B 0,C 180,E1 -23011.873,E2 -23011.873} C_VEL
LIN {X 0,Y 178.186,Z 292.103,A -85,B 0,C 180,E1 -23015.115,E2 -23015.115} C_VEL
LIN {X 0,Y 181.624,Z 287.355,A -85,B 0,C 180,E1 -23018.23,E2 -23018.23} C_VEL
LIN {X 0,Y 185.563,Z 281.07,A -85,B 0,C 180,E1 -23021.234,E2 -23021.234} C_VEL
LIN {X 0,Y 187.425,Z 277.563,A -85,B 0,C 180,E1 -23022.546,E2 -23022.546} C_VEL
LIN {X 0,Y 188.337,Z 272.045,A -85,B 0,C 180,E1 -23024.86,E2 -23024.86} C_VEL
LIN {X 0,Y 188.52,Z 264.14,A -85,B 0,C 180,E1 -23028.048,E2 -23028.048} C_VEL
LIN {X 0,Y 187.721,Z 257.13,A -85,B 0,C 180,E1 -23030.778,E2 -23030.778} C_VEL
LIN {X 0,Y 186.124,Z 250.639,A -85,B 0,C 180,E1 -23033.498,E2 -23033.498} C_VEL
LIN {X 0,Y 184.257,Z 246.107,A -85,B 0,C 180,E1 -23035.627,E2 -23035.627} C_VEL
LIN {X 0,Y 182.32,Z 241.96,A -85,B 0,C 180,E1 -23037.793,E2 -23037.793} C_VEL
LIN {X 0,Y 180.341,Z 237.974,A -85,B 0,C 180,E1 -23040.002,E2 -23040.002} C_VEL
LIN {X 0,Y 178.026,Z 234.336,A -85,B 0,C 180,E1 -23042.477,E2 -23042.477} C_VEL
LIN {X 0,Y 177.782,Z 233.614,A -85,B 0,C 180,E1 -23042.835,E2 -23042.835} C_VEL
LIN {X 0,Y 174.816,Z 231.007,A -85,B 0,C 180,E1 -23045.915,E2 -23045.915} C_VEL
LIN {X 0,Y 173.517,Z 228.323,A -85,B 0,C 180,E1 -23048.005,E2 -23048.005} C_VEL
LIN {X 0,Y 173.446,Z 227.984,A -85,B 0,C 180,E1 -23048.742,E2 -23048.742} C_VEL
LIN {X 0,Y 173.219,Z 227.693,A -85,B 0,C 180,E1 -23053.159,E2 -23053.159} C_VEL
LIN {X 0,Y 173.101,Z 227.795,A -85,B 0,C 180,E1 -23058.956,E2 -23058.956} C_VEL
LIN {X 0,Y 173.125,Z 228.348,A -85,B 0,C 180,E1 -23063.953,E2 -23063.953} C_VEL
LIN {X 0,Y 173.241,Z 228.838,A -85,B 0,C 180,E1 -23066.812,E2 -23066.812} C_VEL
LIN {X 0,Y 173.418,Z 230.092,A -85,B 0,C 180,E1 -23071.794,E2 -23071.794} C_VEL
LIN {X 0,Y 173.708,Z 231.754,A -85,B 0,C 180,E1 -23076.36,E2 -23076.36} C_VEL
LIN {X 0,Y 174.833,Z 234.584,A -85,B 0,C 180,E1 -23078.027,E2 -23078.027} C_VEL
LIN {X 0,Y 177.657,Z 238.327,A -85,B 0,C 180,E1 -23081.163,E2 -23081.163} C_VEL
LIN {X 0,Y 179.428,Z 242.316,A -85,B 0,C 180,E1 -23083.165,E2 -23083.165} C_VEL
LIN {X 0,Y 180.773,Z 244.19,A -85,B 0,C 180,E1 -23084.413,E2 -23084.413} C_VEL
LIN {X 0,Y 183.768,Z 250.543,A -85,B 0,C 180,E1 -23087.476,E2 -23087.476} C_VEL
LIN {X 0,Y 186.562,Z 257.746,A -85,B 0,C 180,E1 -23090.557,E2 -23090.557} C_VEL
LIN {X 0,Y 187.57,Z 261.335,A -85,B 0,C 180,E1 -23091.894,E2 -23091.894} C_VEL
LIN {X 0,Y 187.852,Z 268.721,A -85,B 0,C 180,E1 -23094.15,E2 -23094.15} C_VEL
LIN {X 0,Y 187.176,Z 277.331,A -85,B 0,C 180,E1 -23096.869,E2 -23096.869} C_VEL
LIN {X 0,Y 186.293,Z 282.981,A -85,B 0,C 180,E1 -23098.754,E2 -23098.754} C_VEL
LIN {X 0,Y 184.717,Z 289.238,A -85,B 0,C 180,E1 -23101.059,E2 -23101.059} C_VEL
LIN {X 0,Y 182.753,Z 294.343,A -85,B 0,C 180,E1 -23103.137,E2 -23103.137} C_VEL
LIN {X 0,Y 179.468,Z 299.841,A -85,B 0,C 180,E1 -23105.721,E2 -23105.721} C_VEL
LIN {X 0,Y 176.035,Z 305.025,A -85,B 0,C 180,E1 -23108.942,E2 -23108.942} C_VEL
LIN {X 0,Y 173.284,Z 308.903,A -85,B 0,C 180,E1 -23112.291,E2 -23112.291} C_VEL
LIN {X 0,Y 171.277,Z 311.55,A -85,B 0,C 180,E1 -23115.748,E2 -23115.748} C_VEL
LIN {X 0,Y 170.305,Z 312.623,A -85,B 0,C 180,E1 -23118.093,E2 -23118.093} C_VEL
LIN {X 0,Y 169.623,Z 313.216,A -85,B 0,C 180,E1 -23120.461,E2 -23120.461} C_VEL
LIN {X 0,Y 169.208,Z 313.367,A -85,B 0,C 180,E1 -23122.843,E2 -23122.843} C_VEL
LIN {X 0,Y 169.075,Z 312.787,A -85,B 0,C 180,E1 -23126.064,E2 -23126.064} C_VEL
LIN {X 0,Y 169.239,Z 312.247,A -85,B 0,C 180,E1 -23127.62,E2 -23127.62} C_VEL
LIN {X 0,Y 169.366,Z 310.834,A -85,B 0,C 180,E1 -23130,E2 -23130} C_VEL
LIN {X 0,Y 169.279,Z 307.672,A -85,B 0,C 180,E1 -23133.634,E2 -23133.634} C_VEL
LIN {X 0,Y 169.388,Z 303.092,A -85,B 0,C 180,E1 -23137.151,E2 -23137.151} C_VEL
LIN {X 0,Y 169.865,Z 297.992,A -85,B 0,C 180,E1 -23140.128,E2 -23140.128} C_VEL
LIN {X 0,Y 170.645,Z 291.555,A -85,B 0,C 180,E1 -23143.093,E2 -23143.093} C_VEL
LIN {X 0,Y 171.785,Z 283.449,A -85,B 0,C 180,E1 -23146.031,E2 -23146.031} C_VEL
LIN {X 0,Y 172.741,Z 276.283,A -85,B 0,C 180,E1 -23148.073,E2 -23148.073} C_VEL
LIN {X 0,Y 172.562,Z 267.352,A -85,B 0,C 180,E1 -23150.162,E2 -23150.162} C_VEL
LIN {X 0,Y 172.171,Z 258.365,A -85,B 0,C 180,E1 -23151.869,E2 -23151.869} C_VEL
LIN {X 0,Y 171.727,Z 249.616,A -85,B 0,C 180,E1 -23153.198,E2 -23153.198} C_VEL
LIN {X 0,Y 171.565,Z 246.587,A -85,B 0,C 180,E1 -23153.608,E2 -23153.608} C_VEL
LIN {X 0,Y 170.646,Z 242.936,A -85,B 0,C 180,E1 -23154.183,E2 -23154.183} C_VEL
LIN {X 0,Y 168.938,Z 239.783,A -85,B 0,C 180,E1 -23154.914,E2 -23154.914} C_VEL
LIN {X 0,Y 166.425,Z 236.322,A -85,B 0,C 180,E1 -23156.135,E2 -23156.135} C_VEL
LIN {X 0,Y 164.844,Z 233.941,A -85,B 0,C 180,E1 -23157.471,E2 -23157.471} C_VEL
LIN {X 0,Y 164.617,Z 232.684,A -85,B 0,C 180,E1 -23158.561,E2 -23158.561} C_VEL
LIN {X 0,Y 165.619,Z 229.657,A -85,B 0,C 180,E1 -23161.927,E2 -23161.927} C_VEL
LIN {X 0,Y 165.93,Z 228.349,A -85,B 0,C 180,E1 -23163.41,E2 -23163.41} C_VEL
LIN {X 0,Y 165.5,Z 225.764,A -85,B 0,C 180,E1 -23166.479,E2 -23166.479} C_VEL
LIN {X 0,Y 164.571,Z 220.921,A -85,B 0,C 180,E1 -23172.483,E2 -23172.483} C_VEL
LIN {X 0,Y 164.297,Z 220.828,A -85,B 0,C 180,E1 -23176.808,E2 -23176.808} C_VEL
LIN {X 0,Y 164.298,Z 220.833,A -85,B 0,C 180,E1 -23180.352,E2 -23180.352} C_VEL
LIN {X 0,Y 164.334,Z 220.823,A -85,B 0,C 180,E1 -23184.348,E2 -23184.348} C_VEL
LIN {X 0,Y 164.394,Z 220.819,A -85,B 0,C 180,E1 -23189.133,E2 -23189.133} C_VEL
LIN {X 0,Y 164.411,Z 220.815,A -85,B 0,C 180,E1 -23194.691,E2 -23194.691} C_VEL
LIN {X 0,Y 164.489,Z 220.805,A -85,B 0,C 180,E1 -23200.05,E2 -23200.05} C_VEL
LIN {X 0,Y 164.528,Z 220.803,A -85,B 0,C 180,E1 -23205.148,E2 -23205.148} C_VEL
LIN {X 0,Y 164.771,Z 220.768,A -85,B 0,C 180,E1 -23210.175,E2 -23210.175} C_VEL
LIN {X 0,Y 164.833,Z 220.763,A -85,B 0,C 180,E1 -23212.649,E2 -23212.649} C_VEL
LIN {X 0,Y 165.05,Z 220.733,A -85,B 0,C 180,E1 -23217.557,E2 -23217.557} C_VEL
LIN {X 0,Y 165.297,Z 220.705,A -85,B 0,C 180,E1 -23219.998,E2 -23219.998} C_VEL
LIN {X 0,Y 164.765,Z 220.772,A -85,B 0,C 180,E1 -23224.892,E2 -23224.892} C_VEL
LIN {X 0,Y 164.832,Z 220.762,A -85,B 0,C 180,E1 -23227.347,E2 -23227.347} C_VEL
LIN {X 0,Y 164.704,Z 220.782,A -85,B 0,C 180,E1 -23231.058,E2 -23231.058} C_VEL
LIN {X 0,Y 164.452,Z 220.811,A -85,B 0,C 180,E1 -23237.404,E2 -23237.404} C_VEL
LIN {X 0,Y 164.449,Z 220.812,A -85,B 0,C 180,E1 -23239.99,E2 -23239.99} C_VEL
LIN {X 0,Y 164.385,Z 220.82,A -85,B 0,C 180,E1 -23246.126,E2 -23246.126} C_VEL
LIN {X 0,Y 164.375,Z 220.816,A -85,B 0,C 180,E1 -23251.226,E2 -23251.226} C_VEL
LIN {X 0,Y 164.311,Z 220.829,A -85,B 0,C 180,E1 -23256.782,E2 -23256.782} C_VEL
LIN {X 0,Y 164.297,Z 220.828,A -85,B 0,C 180,E1 -23259.911,E2 -23259.911} C_VEL
LIN {X 0,Y 164.276,Z 220.833,A -85,B 0,C 180,E1 -23263.34,E2 -23263.34} C_VEL
LIN {X 0,Y 164.289,Z 220.83,A -85,B 0,C 180,E1 -23266.807,E2 -23266.807} C_VEL
LIN {X 0,Y 164.291,Z 220.831,A -85,B 0,C 180,E1 -23270.35,E2 -23270.35} C_VEL
LIN {X 0,Y 164.326,Z 220.826,A -85,B 0,C 180,E1 -23274.347,E2 -23274.347} C_VEL
LIN {X 0,Y 164.386,Z 220.819,A -85,B 0,C 180,E1 -23279.133,E2 -23279.133} C_VEL
LIN {X 0,Y 164.411,Z 220.813,A -85,B 0,C 180,E1 -23284.693,E2 -23284.693} C_VEL
LIN {X 0,Y 164.479,Z 220.808,A -85,B 0,C 180,E1 -23290.05,E2 -23290.05} C_VEL
LIN {X 0,Y 164.53,Z 220.801,A -85,B 0,C 180,E1 -23295.149,E2 -23295.149} C_VEL
LIN {X 0,Y 164.802,Z 220.766,A -85,B 0,C 180,E1 -23300.178,E2 -23300.178} C_VEL
LIN {X 0,Y 164.845,Z 220.759,A -85,B 0,C 180,E1 -23302.651,E2 -23302.651} C_VEL
LIN {X 0,Y 165.043,Z 220.737,A -85,B 0,C 180,E1 -23307.559,E2 -23307.559} C_VEL
LIN {X 0,Y 165.288,Z 220.703,A -85,B 0,C 180,E1 -23310,E2 -23310} C_VEL
LIN {X 0,Y 164.762,Z 220.774,A -85,B 0,C 180,E1 -23314.893,E2 -23314.893} C_VEL
LIN {X 0,Y 164.816,Z 220.763,A -85,B 0,C 180,E1 -23317.349,E2 -23317.349} C_VEL
LIN {X 0,Y 164.592,Z 220.795,A -85,B 0,C 180,E1 -23320.875,E2 -23320.875} C_VEL
LIN {X 0,Y 163.798,Z 220.893,A -85,B 0,C 180,E1 -23326.194,E2 -23326.194} C_VEL
LIN {X 0,Y 163.156,Z 223.693,A -85,B 0,C 180,E1 -23330.568,E2 -23330.568} C_VEL
LIN {X 0,Y 163.93,Z 228.422,A -85,B 0,C 180,E1 -23331.206,E2 -23331.206} C_VEL
LIN {X 0,Y 165.329,Z 237.663,A -85,B 0,C 180,E1 -23332.493,E2 -23332.493} C_VEL
LIN {X 0,Y 166.592,Z 247.874,A -85,B 0,C 180,E1 -23334.287,E2 -23334.287} C_VEL
LIN {X 0,Y 167.34,Z 254.953,A -85,B 0,C 180,E1 -23335.832,E2 -23335.832} C_VEL
LIN {X 0,Y 166.147,Z 263.781,A -85,B 0,C 180,E1 -23338.072,E2 -23338.072} C_VEL
LIN {X 0,Y 164.93,Z 271.142,A -85,B 0,C 180,E1 -23340.398,E2 -23340.398} C_VEL
LIN {X 0,Y 164.055,Z 276.738,A -85,B 0,C 180,E1 -23342.542,E2 -23342.542} C_VEL
LIN {X 0,Y 163.178,Z 282.231,A -85,B 0,C 180,E1 -23345.088,E2 -23345.088} C_VEL
LIN {X 0,Y 162.224,Z 288.507,A -85,B 0,C 180,E1 -23348.761,E2 -23348.761} C_VEL
LIN {X 0,Y 161.751,Z 293.041,A -85,B 0,C 180,E1 -23352.388,E2 -23352.388} C_VEL
LIN {X 0,Y 161.735,Z 296.165,A -85,B 0,C 180,E1 -23355.956,E2 -23355.956} C_VEL
LIN {X 0,Y 162.155,Z 298.157,A -85,B 0,C 180,E1 -23359.453,E2 -23359.453} C_VEL
LIN {X 0,Y 163.078,Z 299.123,A -85,B 0,C 180,E1 -23362.893,E2 -23362.893} C_VEL
LIN {X 0,Y 164.501,Z 299.104,A -85,B 0,C 180,E1 -23366.265,E2 -23366.265} C_VEL
LIN {X 0,Y 166.362,Z 298.141,A -85,B 0,C 180,E1 -23369.542,E2 -23369.542} C_VEL
LIN {X 0,Y 168.732,Z 296.199,A -85,B 0,C 180,E1 -23372.734,E2 -23372.734} C_VEL
LIN {X 0,Y 171.498,Z 293.228,A -85,B 0,C 180,E1 -23375.81,E2 -23375.81} C_VEL
LIN {X 0,Y 174.785,Z 289.086,A -85,B 0,C 180,E1 -23378.786,E2 -23378.786} C_VEL
LIN {X 0,Y 178.044,Z 284.386,A -85,B 0,C 180,E1 -23381.326,E2 -23381.326} C_VEL
LIN {X 0,Y 181.379,Z 278.849,A -85,B 0,C 180,E1 -23383.687,E2 -23383.687} C_VEL
LIN {X 0,Y 182.308,Z 273.923,A -85,B 0,C 180,E1 -23385.963,E2 -23385.963} C_VEL
LIN {X 0,Y 182.715,Z 268.443,A -85,B 0,C 180,E1 -23388.352,E2 -23388.352} C_VEL
LIN {X 0,Y 182.446,Z 261.944,A -85,B 0,C 180,E1 -23391.138,E2 -23391.138} C_VEL
LIN {X 0,Y 181.683,Z 257.069,A -85,B 0,C 180,E1 -23393.338,E2 -23393.338} C_VEL
LIN {X 0,Y 180.373,Z 252.577,A -85,B 0,C 180,E1 -23395.533,E2 -23395.533} C_VEL
LIN {X 0,Y 178.118,Z 247.112,A -85,B 0,C 180,E1 -23398.614,E2 -23398.614} C_VEL
LIN {X 0,Y 176.222,Z 243.116,A -85,B 0,C 180,E1 -23401.145,E2 -23401.145} C_VEL
LIN {X 0,Y 174.524,Z 239.85,A -85,B 0,C 180,E1 -23403.466,E2 -23403.466} C_VEL
LIN {X 0,Y 171.767,Z 236.726,A -85,B 0,C 180,E1 -23407.053,E2 -23407.053} C_VEL
LIN {X 0,Y 170.749,Z 234.521,A -85,B 0,C 180,E1 -23408.947,E2 -23408.947} C_VEL
LIN {X 0,Y 167.003,Z 231.396,A -85,B 0,C 180,E1 -23417.766,E2 -23417.766} C_VEL
LIN {X 0,Y 166.624,Z 231.028,A -85,B 0,C 180,E1 -23421.886,E2 -23421.886} C_VEL
LIN {X 0,Y 167.08,Z 232.329,A -85,B 0,C 180,E1 -23426.593,E2 -23426.593} C_VEL
LIN {X 0,Y 171.017,Z 237.956,A -85,B 0,C 180,E1 -23435.509,E2 -23435.509} C_VEL
LIN {X 0,Y 172.272,Z 241.238,A -85,B 0,C 180,E1 -23437.732,E2 -23437.732} C_VEL
LIN {X 0,Y 174.192,Z 244.125,A -85,B 0,C 180,E1 -23440.208,E2 -23440.208} C_VEL
LIN {X 0,Y 177.167,Z 250.318,A -85,B 0,C 180,E1 -23443.967,E2 -23443.967} C_VEL
LIN {X 0,Y 179.751,Z 257.02,A -85,B 0,C 180,E1 -23447.381,E2 -23447.381} C_VEL
LIN {X 0,Y 181.615,Z 262.279,A -85,B 0,C 180,E1 -23449.843,E2 -23449.843} C_VEL
LIN {X 0,Y 182.252,Z 265.125,A -85,B 0,C 180,E1 -23451.015,E2 -23451.015} C_VEL
LIN {X 0,Y 182.168,Z 271.484,A -85,B 0,C 180,E1 -23453.147,E2 -23453.147} C_VEL
LIN {X 0,Y 181.328,Z 278.811,A -85,B 0,C 180,E1 -23455.635,E2 -23455.635} C_VEL
LIN {X 0,Y 179.865,Z 285.685,A -85,B 0,C 180,E1 -23458.164,E2 -23458.164} C_VEL
LIN {X 0,Y 177.511,Z 292.851,A -85,B 0,C 180,E1 -23461.092,E2 -23461.092} C_VEL
LIN {X 0,Y 174.46,Z 298.414,A -85,B 0,C 180,E1 -23463.697,E2 -23463.697} C_VEL
LIN {X 0,Y 170.601,Z 303.814,A -85,B 0,C 180,E1 -23466.961,E2 -23466.961} C_VEL
LIN {X 0,Y 167.386,Z 307.871,A -85,B 0,C 180,E1 -23470.374,E2 -23470.374} C_VEL
LIN {X 0,Y 165.735,Z 309.886,A -85,B 0,C 180,E1 -23472.733,E2 -23472.733} C_VEL
LIN {X 0,Y 164.395,Z 311.428,A -85,B 0,C 180,E1 -23475.138,E2 -23475.138} C_VEL
LIN {X 0,Y 163.338,Z 312.47,A -85,B 0,C 180,E1 -23477.577,E2 -23477.577} C_VEL
LIN {X 0,Y 162.608,Z 312.945,A -85,B 0,C 180,E1 -23480.045,E2 -23480.045} C_VEL
LIN {X 0,Y 162.159,Z 312.966,A -85,B 0,C 180,E1 -23482.53,E2 -23482.53} C_VEL
LIN {X 0,Y 162.008,Z 312.162,A -85,B 0,C 180,E1 -23486.183,E2 -23486.183} C_VEL
LIN {X 0,Y 162.172,Z 311.671,A -85,B 0,C 180,E1 -23487.517,E2 -23487.517} C_VEL
LIN {X 0,Y 162.305,Z 310.194,A -85,B 0,C 180,E1 -23490,E2 -23490} C_VEL
LIN {X 0,Y 162.219,Z 307.117,A -85,B 0,C 180,E1 -23493.531,E2 -23493.531} C_VEL
LIN {X 0,Y 162.263,Z 303.904,A -85,B 0,C 180,E1 -23496.217,E2 -23496.217} C_VEL
LIN {X 0,Y 162.757,Z 297.957,A -85,B 0,C 180,E1 -23499.947,E2 -23499.947} C_VEL
LIN {X 0,Y 163.32,Z 292.979,A -85,B 0,C 180,E1 -23502.425,E2 -23502.425} C_VEL
LIN {X 0,Y 164.177,Z 286.965,A -85,B 0,C 180,E1 -23504.883,E2 -23504.883} C_VEL
LIN {X 0,Y 165.283,Z 279.638,A -85,B 0,C 180,E1 -23507.317,E2 -23507.317} C_VEL
LIN {X 0,Y 165.703,Z 275.321,A -85,B 0,C 180,E1 -23508.549,E2 -23508.549} C_VEL
LIN {X 0,Y 165.507,Z 267.528,A -85,B 0,C 180,E1 -23510.459,E2 -23510.459} C_VEL
LIN {X 0,Y 165.173,Z 258.444,A -85,B 0,C 180,E1 -23512.276,E2 -23512.276} C_VEL
LIN {X 0,Y 164.736,Z 249.238,A -85,B 0,C 180,E1 -23513.743,E2 -23513.743} C_VEL
LIN {X 0,Y 163.962,Z 237.826,A -85,B 0,C 180,E1 -23515.127,E2 -23515.127} C_VEL
LIN {X 0,Y 163.804,Z 235.515,A -85,B 0,C 180,E1 -23515.408,E2 -23515.408} C_VEL
LIN {X 0,Y 164.617,Z 232.684,A -85,B 0,C 180,E1 -23518.561,E2 -23518.561} C_VEL
LIN {X 0,Y 164.628,Z 231.53,A -85,B 0,C 180,E1 -23519.87,E2 -23519.87} C_VEL
LIN {X 0,Y 164.061,Z 230.43,A -85,B 0,C 180,E1 -23521.175,E2 -23521.175} C_VEL
LIN {X 0,Y 161.904,Z 228.383,A -85,B 0,C 180,E1 -23523.774,E2 -23523.774} C_VEL
LIN {X 0,Y 158.468,Z 225.384,A -85,B 0,C 180,E1 -23527.838,E2 -23527.838} C_VEL
LIN {X 0,Y 157.955,Z 224.322,A -85,B 0,C 180,E1 -23529.248,E2 -23529.248} C_VEL
LIN {X 0,Y 157.493,Z 221.679,A -85,B 0,C 180,E1 -23532.845,E2 -23532.845} C_VEL
LIN {X 0,Y 157.209,Z 221.713,A -85,B 0,C 180,E1 -23539.464,E2 -23539.464} C_VEL
LIN {X 0,Y 157.282,Z 221.7,A -85,B 0,C 180,E1 -23544.484,E2 -23544.484} C_VEL
LIN {X 0,Y 157.297,Z 221.705,A -85,B 0,C 180,E1 -23548.095,E2 -23548.095} C_VEL
LIN {X 0,Y 157.319,Z 221.696,A -85,B 0,C 180,E1 -23553.463,E2 -23553.463} C_VEL
LIN {X 0,Y 157.397,Z 221.69,A -85,B 0,C 180,E1 -23559.667,E2 -23559.667} C_VEL
LIN {X 0,Y 157.458,Z 221.682,A -85,B 0,C 180,E1 -23564.464,E2 -23564.464} C_VEL
LIN {X 0,Y 157.693,Z 221.65,A -85,B 0,C 180,E1 -23569.729,E2 -23569.729} C_VEL
LIN {X 0,Y 157.77,Z 221.643,A -85,B 0,C 180,E1 -23572.318,E2 -23572.318} C_VEL
LIN {X 0,Y 158.259,Z 221.581,A -85,B 0,C 180,E1 -23579.998,E2 -23579.998} C_VEL
LIN {X 0,Y 157.768,Z 221.642,A -85,B 0,C 180,E1 -23587.678,E2 -23587.678} C_VEL
LIN {X 0,Y 157.634,Z 221.662,A -85,B 0,C 180,E1 -23591.227,E2 -23591.227} C_VEL
LIN {X 0,Y 157.422,Z 221.683,A -85,B 0,C 180,E1 -23595.535,E2 -23595.535} C_VEL
